HMI tags "2935RS001A01T05"
   "2935RS001A01T05.MSW" : 52809b66-421d-457f-8884-6f7a49d4e247 AT %DB5081.DBX18.0, 500 ms
   "2935RS001A01T05.DefaultText" : TextRef, internal   // Заголовок POPUP окна. При експорте из ECS через скрипт заполняется автоматически, если теги копируются в ручную то требуется в ручную задатать свойство Start Value
   "2935RS001A01T05.BlockInfo" : Array [0..2] of Int AT %DB5081.DBX38.0, 500 ms
   "2935RS001A01T05.StatusWork" : Int AT %DB5081.DBW242, 500 ms
   "2935RS001A01T05.FP_PARAM.DampingTime" : Int AT %DB5081.DBW50, 500 ms
   "2935RS001A01T05.FP_PARAM.Force_Value" : Real AT %DB5081.DBD52, 500 ms
   "2935RS001A01T05.FP_PARAM.Scale_Min" : Real AT %DB5081.DBD56, 500 ms
   "2935RS001A01T05.FP_PARAM.Scale_Max" : Real AT %DB5081.DBD60, 500 ms
   "2935RS001A01T05.FP_PARAM.Gradient" : Real AT %DB5081.DBD64, 500 ms
   "2935RS001A01T05.FP_PARAM.Grad_Pos" : Real AT %DB5081.DBD68, 500 ms
   "2935RS001A01T05.FP_PARAM.Grad_Neg" : Real AT %DB5081.DBD72, 500 ms
   "2935RS001A01T05.FP_PARAM.Grad_X" : Real AT %DB5081.DBD76, 500 ms
   "2935RS001A01T05.FP_PARAM.Gradient_Time_Pre" : Int AT %DB5081.DBW80, 500 ms
   "2935RS001A01T05.FP_PARAM.Gradient_Time_ACC" : Int AT %DB5081.DBW82, 500 ms
   "2935RS001A01T05.FP_PARAM.Alarm_Hyst" : Real AT %DB5081.DBD84, 500 ms
   "2935RS001A01T05.FP_PARAM.AlarmLimit_H3" : Real AT %DB5081.DBD88, 500 ms
   "2935RS001A01T05.FP_PARAM.AlarmLimit_H2" : Real AT %DB5081.DBD92, 500 ms
   "2935RS001A01T05.FP_PARAM.AlarmLimit_H1" : Real AT %DB5081.DBD96, 500 ms
   "2935RS001A01T05.FP_PARAM.AlarmLimit_L1" : Real AT %DB5081.DBD100, 500 ms
   "2935RS001A01T05.FP_PARAM.AlarmLimit_L2" : Real AT %DB5081.DBD104, 500 ms
   "2935RS001A01T05.FP_PARAM.AlarmLimit_L3" : Real AT %DB5081.DBD108, 500 ms
   "2935RS001A01T05.FP_PARAM.AlarmDelay_H3_Pre" : Int AT %DB5081.DBW112, 500 ms
   "2935RS001A01T05.FP_PARAM.AlarmDelay_H3_Acc" : Int AT %DB5081.DBW114, 500 ms
   "2935RS001A01T05.FP_PARAM.AlarmDelay_H2_Pre" : Int AT %DB5081.DBW116, 500 ms
   "2935RS001A01T05.FP_PARAM.AlarmDelay_H2_Acc" : Int AT %DB5081.DBW118, 500 ms
   "2935RS001A01T05.FP_PARAM.AlarmDelay_H1_Pre" : Int AT %DB5081.DBW120, 500 ms
   "2935RS001A01T05.FP_PARAM.AlarmDelay_H1_Acc" : Int AT %DB5081.DBW122, 500 ms
   "2935RS001A01T05.FP_PARAM.AlarmDelay_L1_Pre" : Int AT %DB5081.DBW124, 500 ms
   "2935RS001A01T05.FP_PARAM.AlarmDelay_L1_Acc" : Int AT %DB5081.DBW126, 500 ms
   "2935RS001A01T05.FP_PARAM.AlarmDelay_L2_Pre" : Int AT %DB5081.DBW128, 500 ms
   "2935RS001A01T05.FP_PARAM.AlarmDelay_L2_Acc" : Int AT %DB5081.DBW130, 500 ms
   "2935RS001A01T05.FP_PARAM.AlarmDelay_L3_Pre" : Int AT %DB5081.DBW132, 500 ms
   "2935RS001A01T05.FP_PARAM.AlarmDelay_L3_Acc" : Int AT %DB5081.DBW134, 500 ms
   "2935RS001A01T05.FP_PARAM.OpenLoopDelay_Pre" : Int AT %DB5081.DBW136, 500 ms
   "2935RS001A01T05.FP_PARAM.OpenLoopDelay_Acc" : Int AT %DB5081.DBW138, 500 ms
   "2935RS001A01T05.FP_PARAM.OverRangeDelay_Pre" : Int AT %DB5081.DBW140, 500 ms
   "2935RS001A01T05.FP_PARAM.OverRangeDelay_Acc" : Int AT %DB5081.DBW142, 500 ms
   "2935RS001A01T05.FP_PARAM.AuxLimit_H2_Value" : Real AT %DB5081.DBD144, 500 ms
   "2935RS001A01T05.FP_PARAM.AuxLimit_H1_Value" : Real AT %DB5081.DBD148, 500 ms
   "2935RS001A01T05.FP_PARAM.AuxLimit_L2_Value" : Real AT %DB5081.DBD152, 500 ms
   "2935RS001A01T05.FP_PARAM.AuxLimit_L1_Value" : Real AT %DB5081.DBD156, 500 ms
   "2935RS001A01T05.Unit" : TextRef, internal   // Еденицы измерения При експорте из ECS через скрипт заполняется автоматически, если теги копируются в ручную то требуется задатать свойство Text
   "2935RS001A01T05.Decimals" : TextRef, internal   // Формат отображения При експорте из ECS через скрипт, заполняется автоматически. Если теги копируются в ручную то требуется задатать свойство Text s999999.9
   "2935RS001A01T05.FP_EN.Square" : Bool AT %DB5081.DBX46.0, 500 ms
   "2935RS001A01T05.FP_EN.SquareRoot" : Bool AT %DB5081.DBX46.1, 500 ms
   "2935RS001A01T05.FP_EN.ParentSupress" : Bool AT %DB5081.DBX46.2, 500 ms
   "2935RS001A01T05.FP_EN.ParentSupressUnit" : Bool AT %DB5081.DBX46.3, 500 ms
   "2935RS001A01T05.FP_EN.Force" : Bool AT %DB5081.DBX46.4, 500 ms
   "2935RS001A01T05.FP_EN.Damping" : Bool AT %DB5081.DBX46.5, 500 ms
   "2935RS001A01T05.FP_EN.Gradient_Pos" : Bool AT %DB5081.DBX46.6, 500 ms
   "2935RS001A01T05.FP_EN.Gradient_Neg" : Bool AT %DB5081.DBX46.7, 500 ms
   "2935RS001A01T05.FP_EN.Hysteresis" : Bool AT %DB5081.DBX47.0, 500 ms
   "2935RS001A01T05.FP_EN.Alarm_H3" : Bool AT %DB5081.DBX47.1, 500 ms
   "2935RS001A01T05.FP_EN.Alarm_H2" : Bool AT %DB5081.DBX47.2, 500 ms
   "2935RS001A01T05.FP_EN.Alarm_H1" : Bool AT %DB5081.DBX47.3, 500 ms
   "2935RS001A01T05.FP_EN.Alarm_L1" : Bool AT %DB5081.DBX47.4, 500 ms
   "2935RS001A01T05.FP_EN.Alarm_L2" : Bool AT %DB5081.DBX47.5, 500 ms
   "2935RS001A01T05.FP_EN.Alarm_L3" : Bool AT %DB5081.DBX47.6, 500 ms
   "2935RS001A01T05.FP_EN.AlarmDelay_H3" : Bool AT %DB5081.DBX47.7, 500 ms
   "2935RS001A01T05.FP_EN.AlarmDelay_H2" : Bool AT %DB5081.DBX48.0, 500 ms
   "2935RS001A01T05.FP_EN.AlarmDelay_H1" : Bool AT %DB5081.DBX48.1, 500 ms
   "2935RS001A01T05.FP_EN.AlarmDelay_L1" : Bool AT %DB5081.DBX48.2, 500 ms
   "2935RS001A01T05.FP_EN.AlarmDelay_L2" : Bool AT %DB5081.DBX48.3, 500 ms
   "2935RS001A01T05.FP_EN.AlarmDelay_L3" : Bool AT %DB5081.DBX48.4, 500 ms
   "2935RS001A01T05.FP_EN.ROC_Warn" : Bool AT %DB5081.DBX48.5, 500 ms
   "2935RS001A01T05.FP_EN.U_Range_Warn" : Bool AT %DB5081.DBX48.6, 500 ms
   "2935RS001A01T05.FP_EN.O_Range_Warn" : Bool AT %DB5081.DBX48.7, 500 ms
   "2935RS001A01T05.trend_tag_name" : TextRef, internal   // Еденицы измерения При експорте из ECS через скрипт - заполняется автоматически, если теги копируются в ручную то требуется задатать свойство Text - имя тега для тренда
   "2935RS001A01T05.DQ.AL_H3" : Bool AT %DB5081.DBX16.0, 500 ms
   "2935RS001A01T05.DQ.AL_H2" : Bool AT %DB5081.DBX16.1, 500 ms
   "2935RS001A01T05.DQ.AL_H1" : Bool AT %DB5081.DBX16.2, 500 ms
   "2935RS001A01T05.DQ.AL_L1" : Bool AT %DB5081.DBX16.3, 500 ms
   "2935RS001A01T05.DQ.AL_L2" : Bool AT %DB5081.DBX16.4, 500 ms
   "2935RS001A01T05.DQ.AL_L3" : Bool AT %DB5081.DBX16.5, 500 ms
   "2935RS001A01T05.DQ.SIG_OK" : Bool AT %DB5081.DBX16.6, 500 ms
   "2935RS001A01T05.DQ.LIM_H2" : Bool AT %DB5081.DBX16.7, 500 ms
   "2935RS001A01T05.DQ.LIM_H1" : Bool AT %DB5081.DBX17.0, 500 ms
   "2935RS001A01T05.DQ.LIM_L1" : Bool AT %DB5081.DBX17.1, 500 ms
   "2935RS001A01T05.DQ.LIM_L2" : Bool AT %DB5081.DBX17.2, 500 ms
   "2935RS001A01T05.DQ.GR_P" : Bool AT %DB5081.DBX17.3, 500 ms
   "2935RS001A01T05.DQ.GR_N" : Bool AT %DB5081.DBX17.4, 500 ms
   "2935RS001A01T05.I.IN" : Real AT %DB5081.DBD2, 500 ms
   "2935RS001A01T05.I.SIG_TYPE" : Int AT %DB5081.DBW0, 500 ms
   "2935RS001A01T05.I.FI_BUS" : Byte AT %DB5081.DBB6, 500 ms
   "2935RS001A01T05.DI.U_RANGE" : Bool AT %DB5081.DBX7.0, 500 ms
   "2935RS001A01T05.DI.O_RANGE" : Bool AT %DB5081.DBX7.1, 500 ms
   "2935RS001A01T05.DI.SIG_FAULT" : Bool AT %DB5081.DBX7.2, 500 ms
   "2935RS001A01T05.DI.EnConfig" : Bool AT %DB5081.DBX7.3, 500 ms
   "2935RS001A01T05.DI.AEN" : Bool AT %DB5081.DBX7.4, 500 ms
   "2935RS001A01T05.DI.AL_SUPR" : Bool AT %DB5081.DBX7.5, 500 ms
   "2935RS001A01T05.Q.PV_NORM" : Real AT %DB5081.DBD8, 500 ms
   "2935RS001A01T05.Q.PV_SCAL" : Real AT %DB5081.DBD12, 500 ms
   "2935RS001A01T05.ParentInfo" : TextRef, internal   // Имя родителя для попап окна, вкладка инфо. При експорте из ECS через скрипт заполняется автоматически, если теги копируются в ручную то требуется в ручную задатать свойство Start Value

HMI tags "2940RS001A01F01"
   "2940RS001A01F01.MSW" : 52809b66-421d-457f-8884-6f7a49d4e247 AT %DB5082.DBX18.0, 500 ms
   "2940RS001A01F01.DefaultText" : TextRef, internal   // Заголовок POPUP окна. При експорте из ECS через скрипт заполняется автоматически, если теги копируются в ручную то требуется в ручную задатать свойство Start Value
   "2940RS001A01F01.BlockInfo" : Array [0..2] of Int AT %DB5082.DBX38.0, 500 ms
   "2940RS001A01F01.StatusWork" : Int AT %DB5082.DBW242, 500 ms
   "2940RS001A01F01.FP_PARAM.DampingTime" : Int AT %DB5082.DBW50, 500 ms
   "2940RS001A01F01.FP_PARAM.Force_Value" : Real AT %DB5082.DBD52, 500 ms
   "2940RS001A01F01.FP_PARAM.Scale_Min" : Real AT %DB5082.DBD56, 500 ms
   "2940RS001A01F01.FP_PARAM.Scale_Max" : Real AT %DB5082.DBD60, 500 ms
   "2940RS001A01F01.FP_PARAM.Gradient" : Real AT %DB5082.DBD64, 500 ms
   "2940RS001A01F01.FP_PARAM.Grad_Pos" : Real AT %DB5082.DBD68, 500 ms
   "2940RS001A01F01.FP_PARAM.Grad_Neg" : Real AT %DB5082.DBD72, 500 ms
   "2940RS001A01F01.FP_PARAM.Grad_X" : Real AT %DB5082.DBD76, 500 ms
   "2940RS001A01F01.FP_PARAM.Gradient_Time_Pre" : Int AT %DB5082.DBW80, 500 ms
   "2940RS001A01F01.FP_PARAM.Gradient_Time_ACC" : Int AT %DB5082.DBW82, 500 ms
   "2940RS001A01F01.FP_PARAM.Alarm_Hyst" : Real AT %DB5082.DBD84, 500 ms
   "2940RS001A01F01.FP_PARAM.AlarmLimit_H3" : Real AT %DB5082.DBD88, 500 ms
   "2940RS001A01F01.FP_PARAM.AlarmLimit_H2" : Real AT %DB5082.DBD92, 500 ms
   "2940RS001A01F01.FP_PARAM.AlarmLimit_H1" : Real AT %DB5082.DBD96, 500 ms
   "2940RS001A01F01.FP_PARAM.AlarmLimit_L1" : Real AT %DB5082.DBD100, 500 ms
   "2940RS001A01F01.FP_PARAM.AlarmLimit_L2" : Real AT %DB5082.DBD104, 500 ms
   "2940RS001A01F01.FP_PARAM.AlarmLimit_L3" : Real AT %DB5082.DBD108, 500 ms
   "2940RS001A01F01.FP_PARAM.AlarmDelay_H3_Pre" : Int AT %DB5082.DBW112, 500 ms
   "2940RS001A01F01.FP_PARAM.AlarmDelay_H3_Acc" : Int AT %DB5082.DBW114, 500 ms
   "2940RS001A01F01.FP_PARAM.AlarmDelay_H2_Pre" : Int AT %DB5082.DBW116, 500 ms
   "2940RS001A01F01.FP_PARAM.AlarmDelay_H2_Acc" : Int AT %DB5082.DBW118, 500 ms
   "2940RS001A01F01.FP_PARAM.AlarmDelay_H1_Pre" : Int AT %DB5082.DBW120, 500 ms
   "2940RS001A01F01.FP_PARAM.AlarmDelay_H1_Acc" : Int AT %DB5082.DBW122, 500 ms
   "2940RS001A01F01.FP_PARAM.AlarmDelay_L1_Pre" : Int AT %DB5082.DBW124, 500 ms
   "2940RS001A01F01.FP_PARAM.AlarmDelay_L1_Acc" : Int AT %DB5082.DBW126, 500 ms
   "2940RS001A01F01.FP_PARAM.AlarmDelay_L2_Pre" : Int AT %DB5082.DBW128, 500 ms
   "2940RS001A01F01.FP_PARAM.AlarmDelay_L2_Acc" : Int AT %DB5082.DBW130, 500 ms
   "2940RS001A01F01.FP_PARAM.AlarmDelay_L3_Pre" : Int AT %DB5082.DBW132, 500 ms
   "2940RS001A01F01.FP_PARAM.AlarmDelay_L3_Acc" : Int AT %DB5082.DBW134, 500 ms
   "2940RS001A01F01.FP_PARAM.OpenLoopDelay_Pre" : Int AT %DB5082.DBW136, 500 ms
   "2940RS001A01F01.FP_PARAM.OpenLoopDelay_Acc" : Int AT %DB5082.DBW138, 500 ms
   "2940RS001A01F01.FP_PARAM.OverRangeDelay_Pre" : Int AT %DB5082.DBW140, 500 ms
   "2940RS001A01F01.FP_PARAM.OverRangeDelay_Acc" : Int AT %DB5082.DBW142, 500 ms
   "2940RS001A01F01.FP_PARAM.AuxLimit_H2_Value" : Real AT %DB5082.DBD144, 500 ms
   "2940RS001A01F01.FP_PARAM.AuxLimit_H1_Value" : Real AT %DB5082.DBD148, 500 ms
   "2940RS001A01F01.FP_PARAM.AuxLimit_L2_Value" : Real AT %DB5082.DBD152, 500 ms
   "2940RS001A01F01.FP_PARAM.AuxLimit_L1_Value" : Real AT %DB5082.DBD156, 500 ms
   "2940RS001A01F01.Unit" : TextRef, internal   // Еденицы измерения При експорте из ECS через скрипт заполняется автоматически, если теги копируются в ручную то требуется задатать свойство Text
   "2940RS001A01F01.Decimals" : TextRef, internal   // Формат отображения При експорте из ECS через скрипт, заполняется автоматически. Если теги копируются в ручную то требуется задатать свойство Text s999999.9
   "2940RS001A01F01.FP_EN.Square" : Bool AT %DB5082.DBX46.0, 500 ms
   "2940RS001A01F01.FP_EN.SquareRoot" : Bool AT %DB5082.DBX46.1, 500 ms
   "2940RS001A01F01.FP_EN.ParentSupress" : Bool AT %DB5082.DBX46.2, 500 ms
   "2940RS001A01F01.FP_EN.ParentSupressUnit" : Bool AT %DB5082.DBX46.3, 500 ms
   "2940RS001A01F01.FP_EN.Force" : Bool AT %DB5082.DBX46.4, 500 ms
   "2940RS001A01F01.FP_EN.Damping" : Bool AT %DB5082.DBX46.5, 500 ms
   "2940RS001A01F01.FP_EN.Gradient_Pos" : Bool AT %DB5082.DBX46.6, 500 ms
   "2940RS001A01F01.FP_EN.Gradient_Neg" : Bool AT %DB5082.DBX46.7, 500 ms
   "2940RS001A01F01.FP_EN.Hysteresis" : Bool AT %DB5082.DBX47.0, 500 ms
   "2940RS001A01F01.FP_EN.Alarm_H3" : Bool AT %DB5082.DBX47.1, 500 ms
   "2940RS001A01F01.FP_EN.Alarm_H2" : Bool AT %DB5082.DBX47.2, 500 ms
   "2940RS001A01F01.FP_EN.Alarm_H1" : Bool AT %DB5082.DBX47.3, 500 ms
   "2940RS001A01F01.FP_EN.Alarm_L1" : Bool AT %DB5082.DBX47.4, 500 ms
   "2940RS001A01F01.FP_EN.Alarm_L2" : Bool AT %DB5082.DBX47.5, 500 ms
   "2940RS001A01F01.FP_EN.Alarm_L3" : Bool AT %DB5082.DBX47.6, 500 ms
   "2940RS001A01F01.FP_EN.AlarmDelay_H3" : Bool AT %DB5082.DBX47.7, 500 ms
   "2940RS001A01F01.FP_EN.AlarmDelay_H2" : Bool AT %DB5082.DBX48.0, 500 ms
   "2940RS001A01F01.FP_EN.AlarmDelay_H1" : Bool AT %DB5082.DBX48.1, 500 ms
   "2940RS001A01F01.FP_EN.AlarmDelay_L1" : Bool AT %DB5082.DBX48.2, 500 ms
   "2940RS001A01F01.FP_EN.AlarmDelay_L2" : Bool AT %DB5082.DBX48.3, 500 ms
   "2940RS001A01F01.FP_EN.AlarmDelay_L3" : Bool AT %DB5082.DBX48.4, 500 ms
   "2940RS001A01F01.FP_EN.ROC_Warn" : Bool AT %DB5082.DBX48.5, 500 ms
   "2940RS001A01F01.FP_EN.U_Range_Warn" : Bool AT %DB5082.DBX48.6, 500 ms
   "2940RS001A01F01.FP_EN.O_Range_Warn" : Bool AT %DB5082.DBX48.7, 500 ms
   "2940RS001A01F01.trend_tag_name" : TextRef, internal   // Еденицы измерения При експорте из ECS через скрипт - заполняется автоматически, если теги копируются в ручную то требуется задатать свойство Text - имя тега для тренда
   "2940RS001A01F01.DQ.AL_H3" : Bool AT %DB5082.DBX16.0, 500 ms
   "2940RS001A01F01.DQ.AL_H2" : Bool AT %DB5082.DBX16.1, 500 ms
   "2940RS001A01F01.DQ.AL_H1" : Bool AT %DB5082.DBX16.2, 500 ms
   "2940RS001A01F01.DQ.AL_L1" : Bool AT %DB5082.DBX16.3, 500 ms
   "2940RS001A01F01.DQ.AL_L2" : Bool AT %DB5082.DBX16.4, 500 ms
   "2940RS001A01F01.DQ.AL_L3" : Bool AT %DB5082.DBX16.5, 500 ms
   "2940RS001A01F01.DQ.SIG_OK" : Bool AT %DB5082.DBX16.6, 500 ms
   "2940RS001A01F01.DQ.LIM_H2" : Bool AT %DB5082.DBX16.7, 500 ms
   "2940RS001A01F01.DQ.LIM_H1" : Bool AT %DB5082.DBX17.0, 500 ms
   "2940RS001A01F01.DQ.LIM_L1" : Bool AT %DB5082.DBX17.1, 500 ms
   "2940RS001A01F01.DQ.LIM_L2" : Bool AT %DB5082.DBX17.2, 500 ms
   "2940RS001A01F01.DQ.GR_P" : Bool AT %DB5082.DBX17.3, 500 ms
   "2940RS001A01F01.DQ.GR_N" : Bool AT %DB5082.DBX17.4, 500 ms
   "2940RS001A01F01.I.IN" : Real AT %DB5082.DBD2, 500 ms
   "2940RS001A01F01.I.SIG_TYPE" : Int AT %DB5082.DBW0, 500 ms
   "2940RS001A01F01.I.FI_BUS" : Byte AT %DB5082.DBB6, 500 ms
   "2940RS001A01F01.DI.U_RANGE" : Bool AT %DB5082.DBX7.0, 500 ms
   "2940RS001A01F01.DI.O_RANGE" : Bool AT %DB5082.DBX7.1, 500 ms
   "2940RS001A01F01.DI.SIG_FAULT" : Bool AT %DB5082.DBX7.2, 500 ms
   "2940RS001A01F01.DI.EnConfig" : Bool AT %DB5082.DBX7.3, 500 ms
   "2940RS001A01F01.DI.AEN" : Bool AT %DB5082.DBX7.4, 500 ms
   "2940RS001A01F01.DI.AL_SUPR" : Bool AT %DB5082.DBX7.5, 500 ms
   "2940RS001A01F01.Q.PV_NORM" : Real AT %DB5082.DBD8, 500 ms
   "2940RS001A01F01.Q.PV_SCAL" : Real AT %DB5082.DBD12, 500 ms
   "2940RS001A01F01.ParentInfo" : TextRef, internal   // Имя родителя для попап окна, вкладка инфо. При експорте из ECS через скрипт заполняется автоматически, если теги копируются в ручную то требуется в ручную задатать свойство Start Value

HMI tags "2940RS001A01L01"
   "2940RS001A01L01.MSW" : 52809b66-421d-457f-8884-6f7a49d4e247 AT %DB5083.DBX18.0, 500 ms
   "2940RS001A01L01.DefaultText" : TextRef, internal   // Заголовок POPUP окна. При експорте из ECS через скрипт заполняется автоматически, если теги копируются в ручную то требуется в ручную задатать свойство Start Value
   "2940RS001A01L01.BlockInfo" : Array [0..2] of Int AT %DB5083.DBX38.0, 500 ms
   "2940RS001A01L01.StatusWork" : Int AT %DB5083.DBW242, 500 ms
   "2940RS001A01L01.FP_PARAM.DampingTime" : Int AT %DB5083.DBW50, 500 ms
   "2940RS001A01L01.FP_PARAM.Force_Value" : Real AT %DB5083.DBD52, 500 ms
   "2940RS001A01L01.FP_PARAM.Scale_Min" : Real AT %DB5083.DBD56, 500 ms
   "2940RS001A01L01.FP_PARAM.Scale_Max" : Real AT %DB5083.DBD60, 500 ms
   "2940RS001A01L01.FP_PARAM.Gradient" : Real AT %DB5083.DBD64, 500 ms
   "2940RS001A01L01.FP_PARAM.Grad_Pos" : Real AT %DB5083.DBD68, 500 ms
   "2940RS001A01L01.FP_PARAM.Grad_Neg" : Real AT %DB5083.DBD72, 500 ms
   "2940RS001A01L01.FP_PARAM.Grad_X" : Real AT %DB5083.DBD76, 500 ms
   "2940RS001A01L01.FP_PARAM.Gradient_Time_Pre" : Int AT %DB5083.DBW80, 500 ms
   "2940RS001A01L01.FP_PARAM.Gradient_Time_ACC" : Int AT %DB5083.DBW82, 500 ms
   "2940RS001A01L01.FP_PARAM.Alarm_Hyst" : Real AT %DB5083.DBD84, 500 ms
   "2940RS001A01L01.FP_PARAM.AlarmLimit_H3" : Real AT %DB5083.DBD88, 500 ms
   "2940RS001A01L01.FP_PARAM.AlarmLimit_H2" : Real AT %DB5083.DBD92, 500 ms
   "2940RS001A01L01.FP_PARAM.AlarmLimit_H1" : Real AT %DB5083.DBD96, 500 ms
   "2940RS001A01L01.FP_PARAM.AlarmLimit_L1" : Real AT %DB5083.DBD100, 500 ms
   "2940RS001A01L01.FP_PARAM.AlarmLimit_L2" : Real AT %DB5083.DBD104, 500 ms
   "2940RS001A01L01.FP_PARAM.AlarmLimit_L3" : Real AT %DB5083.DBD108, 500 ms
   "2940RS001A01L01.FP_PARAM.AlarmDelay_H3_Pre" : Int AT %DB5083.DBW112, 500 ms
   "2940RS001A01L01.FP_PARAM.AlarmDelay_H3_Acc" : Int AT %DB5083.DBW114, 500 ms
   "2940RS001A01L01.FP_PARAM.AlarmDelay_H2_Pre" : Int AT %DB5083.DBW116, 500 ms
   "2940RS001A01L01.FP_PARAM.AlarmDelay_H2_Acc" : Int AT %DB5083.DBW118, 500 ms
   "2940RS001A01L01.FP_PARAM.AlarmDelay_H1_Pre" : Int AT %DB5083.DBW120, 500 ms
   "2940RS001A01L01.FP_PARAM.AlarmDelay_H1_Acc" : Int AT %DB5083.DBW122, 500 ms
   "2940RS001A01L01.FP_PARAM.AlarmDelay_L1_Pre" : Int AT %DB5083.DBW124, 500 ms
   "2940RS001A01L01.FP_PARAM.AlarmDelay_L1_Acc" : Int AT %DB5083.DBW126, 500 ms
   "2940RS001A01L01.FP_PARAM.AlarmDelay_L2_Pre" : Int AT %DB5083.DBW128, 500 ms
   "2940RS001A01L01.FP_PARAM.AlarmDelay_L2_Acc" : Int AT %DB5083.DBW130, 500 ms
   "2940RS001A01L01.FP_PARAM.AlarmDelay_L3_Pre" : Int AT %DB5083.DBW132, 500 ms
   "2940RS001A01L01.FP_PARAM.AlarmDelay_L3_Acc" : Int AT %DB5083.DBW134, 500 ms
   "2940RS001A01L01.FP_PARAM.OpenLoopDelay_Pre" : Int AT %DB5083.DBW136, 500 ms
   "2940RS001A01L01.FP_PARAM.OpenLoopDelay_Acc" : Int AT %DB5083.DBW138, 500 ms
   "2940RS001A01L01.FP_PARAM.OverRangeDelay_Pre" : Int AT %DB5083.DBW140, 500 ms
   "2940RS001A01L01.FP_PARAM.OverRangeDelay_Acc" : Int AT %DB5083.DBW142, 500 ms
   "2940RS001A01L01.FP_PARAM.AuxLimit_H2_Value" : Real AT %DB5083.DBD144, 500 ms
   "2940RS001A01L01.FP_PARAM.AuxLimit_H1_Value" : Real AT %DB5083.DBD148, 500 ms
   "2940RS001A01L01.FP_PARAM.AuxLimit_L2_Value" : Real AT %DB5083.DBD152, 500 ms
   "2940RS001A01L01.FP_PARAM.AuxLimit_L1_Value" : Real AT %DB5083.DBD156, 500 ms
   "2940RS001A01L01.Unit" : TextRef, internal   // Еденицы измерения При експорте из ECS через скрипт заполняется автоматически, если теги копируются в ручную то требуется задатать свойство Text
   "2940RS001A01L01.Decimals" : TextRef, internal   // Формат отображения При експорте из ECS через скрипт, заполняется автоматически. Если теги копируются в ручную то требуется задатать свойство Text s999999.9
   "2940RS001A01L01.FP_EN.Square" : Bool AT %DB5083.DBX46.0, 500 ms
   "2940RS001A01L01.FP_EN.SquareRoot" : Bool AT %DB5083.DBX46.1, 500 ms
   "2940RS001A01L01.FP_EN.ParentSupress" : Bool AT %DB5083.DBX46.2, 500 ms
   "2940RS001A01L01.FP_EN.ParentSupressUnit" : Bool AT %DB5083.DBX46.3, 500 ms
   "2940RS001A01L01.FP_EN.Force" : Bool AT %DB5083.DBX46.4, 500 ms
   "2940RS001A01L01.FP_EN.Damping" : Bool AT %DB5083.DBX46.5, 500 ms
   "2940RS001A01L01.FP_EN.Gradient_Pos" : Bool AT %DB5083.DBX46.6, 500 ms
   "2940RS001A01L01.FP_EN.Gradient_Neg" : Bool AT %DB5083.DBX46.7, 500 ms
   "2940RS001A01L01.FP_EN.Hysteresis" : Bool AT %DB5083.DBX47.0, 500 ms
   "2940RS001A01L01.FP_EN.Alarm_H3" : Bool AT %DB5083.DBX47.1, 500 ms
   "2940RS001A01L01.FP_EN.Alarm_H2" : Bool AT %DB5083.DBX47.2, 500 ms
   "2940RS001A01L01.FP_EN.Alarm_H1" : Bool AT %DB5083.DBX47.3, 500 ms
   "2940RS001A01L01.FP_EN.Alarm_L1" : Bool AT %DB5083.DBX47.4, 500 ms
   "2940RS001A01L01.FP_EN.Alarm_L2" : Bool AT %DB5083.DBX47.5, 500 ms
   "2940RS001A01L01.FP_EN.Alarm_L3" : Bool AT %DB5083.DBX47.6, 500 ms
   "2940RS001A01L01.FP_EN.AlarmDelay_H3" : Bool AT %DB5083.DBX47.7, 500 ms
   "2940RS001A01L01.FP_EN.AlarmDelay_H2" : Bool AT %DB5083.DBX48.0, 500 ms
   "2940RS001A01L01.FP_EN.AlarmDelay_H1" : Bool AT %DB5083.DBX48.1, 500 ms
   "2940RS001A01L01.FP_EN.AlarmDelay_L1" : Bool AT %DB5083.DBX48.2, 500 ms
   "2940RS001A01L01.FP_EN.AlarmDelay_L2" : Bool AT %DB5083.DBX48.3, 500 ms
   "2940RS001A01L01.FP_EN.AlarmDelay_L3" : Bool AT %DB5083.DBX48.4, 500 ms
   "2940RS001A01L01.FP_EN.ROC_Warn" : Bool AT %DB5083.DBX48.5, 500 ms
   "2940RS001A01L01.FP_EN.U_Range_Warn" : Bool AT %DB5083.DBX48.6, 500 ms
   "2940RS001A01L01.FP_EN.O_Range_Warn" : Bool AT %DB5083.DBX48.7, 500 ms
   "2940RS001A01L01.trend_tag_name" : TextRef, internal   // Еденицы измерения При експорте из ECS через скрипт - заполняется автоматически, если теги копируются в ручную то требуется задатать свойство Text - имя тега для тренда
   "2940RS001A01L01.DQ.AL_H3" : Bool AT %DB5083.DBX16.0, 500 ms
   "2940RS001A01L01.DQ.AL_H2" : Bool AT %DB5083.DBX16.1, 500 ms
   "2940RS001A01L01.DQ.AL_H1" : Bool AT %DB5083.DBX16.2, 500 ms
   "2940RS001A01L01.DQ.AL_L1" : Bool AT %DB5083.DBX16.3, 500 ms
   "2940RS001A01L01.DQ.AL_L2" : Bool AT %DB5083.DBX16.4, 500 ms
   "2940RS001A01L01.DQ.AL_L3" : Bool AT %DB5083.DBX16.5, 500 ms
   "2940RS001A01L01.DQ.SIG_OK" : Bool AT %DB5083.DBX16.6, 500 ms
   "2940RS001A01L01.DQ.LIM_H2" : Bool AT %DB5083.DBX16.7, 500 ms
   "2940RS001A01L01.DQ.LIM_H1" : Bool AT %DB5083.DBX17.0, 500 ms
   "2940RS001A01L01.DQ.LIM_L1" : Bool AT %DB5083.DBX17.1, 500 ms
   "2940RS001A01L01.DQ.LIM_L2" : Bool AT %DB5083.DBX17.2, 500 ms
   "2940RS001A01L01.DQ.GR_P" : Bool AT %DB5083.DBX17.3, 500 ms
   "2940RS001A01L01.DQ.GR_N" : Bool AT %DB5083.DBX17.4, 500 ms
   "2940RS001A01L01.I.IN" : Real AT %DB5083.DBD2, 500 ms
   "2940RS001A01L01.I.SIG_TYPE" : Int AT %DB5083.DBW0, 500 ms
   "2940RS001A01L01.I.FI_BUS" : Byte AT %DB5083.DBB6, 500 ms
   "2940RS001A01L01.DI.U_RANGE" : Bool AT %DB5083.DBX7.0, 500 ms
   "2940RS001A01L01.DI.O_RANGE" : Bool AT %DB5083.DBX7.1, 500 ms
   "2940RS001A01L01.DI.SIG_FAULT" : Bool AT %DB5083.DBX7.2, 500 ms
   "2940RS001A01L01.DI.EnConfig" : Bool AT %DB5083.DBX7.3, 500 ms
   "2940RS001A01L01.DI.AEN" : Bool AT %DB5083.DBX7.4, 500 ms
   "2940RS001A01L01.DI.AL_SUPR" : Bool AT %DB5083.DBX7.5, 500 ms
   "2940RS001A01L01.Q.PV_NORM" : Real AT %DB5083.DBD8, 500 ms
   "2940RS001A01L01.Q.PV_SCAL" : Real AT %DB5083.DBD12, 500 ms
   "2940RS001A01L01.ParentInfo" : TextRef, internal   // Имя родителя для попап окна, вкладка инфо. При експорте из ECS через скрипт заполняется автоматически, если теги копируются в ручную то требуется в ручную задатать свойство Start Value

HMI tags "2940RS001A01T01"
   "2940RS001A01T01.MSW" : 52809b66-421d-457f-8884-6f7a49d4e247 AT %DB5084.DBX18.0, 500 ms
   "2940RS001A01T01.DefaultText" : TextRef, internal   // Заголовок POPUP окна. При експорте из ECS через скрипт заполняется автоматически, если теги копируются в ручную то требуется в ручную задатать свойство Start Value
   "2940RS001A01T01.BlockInfo" : Array [0..2] of Int AT %DB5084.DBX38.0, 500 ms
   "2940RS001A01T01.StatusWork" : Int AT %DB5084.DBW242, 500 ms
   "2940RS001A01T01.FP_PARAM.DampingTime" : Int AT %DB5084.DBW50, 500 ms
   "2940RS001A01T01.FP_PARAM.Force_Value" : Real AT %DB5084.DBD52, 500 ms
   "2940RS001A01T01.FP_PARAM.Scale_Min" : Real AT %DB5084.DBD56, 500 ms
   "2940RS001A01T01.FP_PARAM.Scale_Max" : Real AT %DB5084.DBD60, 500 ms
   "2940RS001A01T01.FP_PARAM.Gradient" : Real AT %DB5084.DBD64, 500 ms
   "2940RS001A01T01.FP_PARAM.Grad_Pos" : Real AT %DB5084.DBD68, 500 ms
   "2940RS001A01T01.FP_PARAM.Grad_Neg" : Real AT %DB5084.DBD72, 500 ms
   "2940RS001A01T01.FP_PARAM.Grad_X" : Real AT %DB5084.DBD76, 500 ms
   "2940RS001A01T01.FP_PARAM.Gradient_Time_Pre" : Int AT %DB5084.DBW80, 500 ms
   "2940RS001A01T01.FP_PARAM.Gradient_Time_ACC" : Int AT %DB5084.DBW82, 500 ms
   "2940RS001A01T01.FP_PARAM.Alarm_Hyst" : Real AT %DB5084.DBD84, 500 ms
   "2940RS001A01T01.FP_PARAM.AlarmLimit_H3" : Real AT %DB5084.DBD88, 500 ms
   "2940RS001A01T01.FP_PARAM.AlarmLimit_H2" : Real AT %DB5084.DBD92, 500 ms
   "2940RS001A01T01.FP_PARAM.AlarmLimit_H1" : Real AT %DB5084.DBD96, 500 ms
   "2940RS001A01T01.FP_PARAM.AlarmLimit_L1" : Real AT %DB5084.DBD100, 500 ms
   "2940RS001A01T01.FP_PARAM.AlarmLimit_L2" : Real AT %DB5084.DBD104, 500 ms
   "2940RS001A01T01.FP_PARAM.AlarmLimit_L3" : Real AT %DB5084.DBD108, 500 ms
   "2940RS001A01T01.FP_PARAM.AlarmDelay_H3_Pre" : Int AT %DB5084.DBW112, 500 ms
   "2940RS001A01T01.FP_PARAM.AlarmDelay_H3_Acc" : Int AT %DB5084.DBW114, 500 ms
   "2940RS001A01T01.FP_PARAM.AlarmDelay_H2_Pre" : Int AT %DB5084.DBW116, 500 ms
   "2940RS001A01T01.FP_PARAM.AlarmDelay_H2_Acc" : Int AT %DB5084.DBW118, 500 ms
   "2940RS001A01T01.FP_PARAM.AlarmDelay_H1_Pre" : Int AT %DB5084.DBW120, 500 ms
   "2940RS001A01T01.FP_PARAM.AlarmDelay_H1_Acc" : Int AT %DB5084.DBW122, 500 ms
   "2940RS001A01T01.FP_PARAM.AlarmDelay_L1_Pre" : Int AT %DB5084.DBW124, 500 ms
   "2940RS001A01T01.FP_PARAM.AlarmDelay_L1_Acc" : Int AT %DB5084.DBW126, 500 ms
   "2940RS001A01T01.FP_PARAM.AlarmDelay_L2_Pre" : Int AT %DB5084.DBW128, 500 ms
   "2940RS001A01T01.FP_PARAM.AlarmDelay_L2_Acc" : Int AT %DB5084.DBW130, 500 ms
   "2940RS001A01T01.FP_PARAM.AlarmDelay_L3_Pre" : Int AT %DB5084.DBW132, 500 ms
   "2940RS001A01T01.FP_PARAM.AlarmDelay_L3_Acc" : Int AT %DB5084.DBW134, 500 ms
   "2940RS001A01T01.FP_PARAM.OpenLoopDelay_Pre" : Int AT %DB5084.DBW136, 500 ms
   "2940RS001A01T01.FP_PARAM.OpenLoopDelay_Acc" : Int AT %DB5084.DBW138, 500 ms
   "2940RS001A01T01.FP_PARAM.OverRangeDelay_Pre" : Int AT %DB5084.DBW140, 500 ms
   "2940RS001A01T01.FP_PARAM.OverRangeDelay_Acc" : Int AT %DB5084.DBW142, 500 ms
   "2940RS001A01T01.FP_PARAM.AuxLimit_H2_Value" : Real AT %DB5084.DBD144, 500 ms
   "2940RS001A01T01.FP_PARAM.AuxLimit_H1_Value" : Real AT %DB5084.DBD148, 500 ms
   "2940RS001A01T01.FP_PARAM.AuxLimit_L2_Value" : Real AT %DB5084.DBD152, 500 ms
   "2940RS001A01T01.FP_PARAM.AuxLimit_L1_Value" : Real AT %DB5084.DBD156, 500 ms
   "2940RS001A01T01.Unit" : TextRef, internal   // Еденицы измерения При експорте из ECS через скрипт заполняется автоматически, если теги копируются в ручную то требуется задатать свойство Text
   "2940RS001A01T01.Decimals" : TextRef, internal   // Формат отображения При експорте из ECS через скрипт, заполняется автоматически. Если теги копируются в ручную то требуется задатать свойство Text s999999.9
   "2940RS001A01T01.FP_EN.Square" : Bool AT %DB5084.DBX46.0, 500 ms
   "2940RS001A01T01.FP_EN.SquareRoot" : Bool AT %DB5084.DBX46.1, 500 ms
   "2940RS001A01T01.FP_EN.ParentSupress" : Bool AT %DB5084.DBX46.2, 500 ms
   "2940RS001A01T01.FP_EN.ParentSupressUnit" : Bool AT %DB5084.DBX46.3, 500 ms
   "2940RS001A01T01.FP_EN.Force" : Bool AT %DB5084.DBX46.4, 500 ms
   "2940RS001A01T01.FP_EN.Damping" : Bool AT %DB5084.DBX46.5, 500 ms
   "2940RS001A01T01.FP_EN.Gradient_Pos" : Bool AT %DB5084.DBX46.6, 500 ms
   "2940RS001A01T01.FP_EN.Gradient_Neg" : Bool AT %DB5084.DBX46.7, 500 ms
   "2940RS001A01T01.FP_EN.Hysteresis" : Bool AT %DB5084.DBX47.0, 500 ms
   "2940RS001A01T01.FP_EN.Alarm_H3" : Bool AT %DB5084.DBX47.1, 500 ms
   "2940RS001A01T01.FP_EN.Alarm_H2" : Bool AT %DB5084.DBX47.2, 500 ms
   "2940RS001A01T01.FP_EN.Alarm_H1" : Bool AT %DB5084.DBX47.3, 500 ms
   "2940RS001A01T01.FP_EN.Alarm_L1" : Bool AT %DB5084.DBX47.4, 500 ms
   "2940RS001A01T01.FP_EN.Alarm_L2" : Bool AT %DB5084.DBX47.5, 500 ms
   "2940RS001A01T01.FP_EN.Alarm_L3" : Bool AT %DB5084.DBX47.6, 500 ms
   "2940RS001A01T01.FP_EN.AlarmDelay_H3" : Bool AT %DB5084.DBX47.7, 500 ms
   "2940RS001A01T01.FP_EN.AlarmDelay_H2" : Bool AT %DB5084.DBX48.0, 500 ms
   "2940RS001A01T01.FP_EN.AlarmDelay_H1" : Bool AT %DB5084.DBX48.1, 500 ms
   "2940RS001A01T01.FP_EN.AlarmDelay_L1" : Bool AT %DB5084.DBX48.2, 500 ms
   "2940RS001A01T01.FP_EN.AlarmDelay_L2" : Bool AT %DB5084.DBX48.3, 500 ms
   "2940RS001A01T01.FP_EN.AlarmDelay_L3" : Bool AT %DB5084.DBX48.4, 500 ms
   "2940RS001A01T01.FP_EN.ROC_Warn" : Bool AT %DB5084.DBX48.5, 500 ms
   "2940RS001A01T01.FP_EN.U_Range_Warn" : Bool AT %DB5084.DBX48.6, 500 ms
   "2940RS001A01T01.FP_EN.O_Range_Warn" : Bool AT %DB5084.DBX48.7, 500 ms
   "2940RS001A01T01.trend_tag_name" : TextRef, internal   // Еденицы измерения При експорте из ECS через скрипт - заполняется автоматически, если теги копируются в ручную то требуется задатать свойство Text - имя тега для тренда
   "2940RS001A01T01.DQ.AL_H3" : Bool AT %DB5084.DBX16.0, 500 ms
   "2940RS001A01T01.DQ.AL_H2" : Bool AT %DB5084.DBX16.1, 500 ms
   "2940RS001A01T01.DQ.AL_H1" : Bool AT %DB5084.DBX16.2, 500 ms
   "2940RS001A01T01.DQ.AL_L1" : Bool AT %DB5084.DBX16.3, 500 ms
   "2940RS001A01T01.DQ.AL_L2" : Bool AT %DB5084.DBX16.4, 500 ms
   "2940RS001A01T01.DQ.AL_L3" : Bool AT %DB5084.DBX16.5, 500 ms
   "2940RS001A01T01.DQ.SIG_OK" : Bool AT %DB5084.DBX16.6, 500 ms
   "2940RS001A01T01.DQ.LIM_H2" : Bool AT %DB5084.DBX16.7, 500 ms
   "2940RS001A01T01.DQ.LIM_H1" : Bool AT %DB5084.DBX17.0, 500 ms
   "2940RS001A01T01.DQ.LIM_L1" : Bool AT %DB5084.DBX17.1, 500 ms
   "2940RS001A01T01.DQ.LIM_L2" : Bool AT %DB5084.DBX17.2, 500 ms
   "2940RS001A01T01.DQ.GR_P" : Bool AT %DB5084.DBX17.3, 500 ms
   "2940RS001A01T01.DQ.GR_N" : Bool AT %DB5084.DBX17.4, 500 ms
   "2940RS001A01T01.I.IN" : Real AT %DB5084.DBD2, 500 ms
   "2940RS001A01T01.I.SIG_TYPE" : Int AT %DB5084.DBW0, 500 ms
   "2940RS001A01T01.I.FI_BUS" : Byte AT %DB5084.DBB6, 500 ms
   "2940RS001A01T01.DI.U_RANGE" : Bool AT %DB5084.DBX7.0, 500 ms
   "2940RS001A01T01.DI.O_RANGE" : Bool AT %DB5084.DBX7.1, 500 ms
   "2940RS001A01T01.DI.SIG_FAULT" : Bool AT %DB5084.DBX7.2, 500 ms
   "2940RS001A01T01.DI.EnConfig" : Bool AT %DB5084.DBX7.3, 500 ms
   "2940RS001A01T01.DI.AEN" : Bool AT %DB5084.DBX7.4, 500 ms
   "2940RS001A01T01.DI.AL_SUPR" : Bool AT %DB5084.DBX7.5, 500 ms
   "2940RS001A01T01.Q.PV_NORM" : Real AT %DB5084.DBD8, 500 ms
   "2940RS001A01T01.Q.PV_SCAL" : Real AT %DB5084.DBD12, 500 ms
   "2940RS001A01T01.ParentInfo" : TextRef, internal   // Имя родителя для попап окна, вкладка инфо. При експорте из ECS через скрипт заполняется автоматически, если теги копируются в ручную то требуется в ручную задатать свойство Start Value

HMI tags "2940RS001N01T01"
   "2940RS001N01T01.MSW" : 52809b66-421d-457f-8884-6f7a49d4e247 AT %DB5304.DBX18.0, 500 ms
   "2940RS001N01T01.DefaultText" : TextRef, internal   // Заголовок POPUP окна. При експорте из ECS через скрипт заполняется автоматически, если теги копируются в ручную то требуется в ручную задатать свойство Start Value
   "2940RS001N01T01.BlockInfo" : Array [0..2] of Int AT %DB5304.DBX38.0, 500 ms
   "2940RS001N01T01.StatusWork" : Int AT %DB5304.DBW242, 500 ms
   "2940RS001N01T01.FP_PARAM.DampingTime" : Int AT %DB5304.DBW50, 500 ms
   "2940RS001N01T01.FP_PARAM.Force_Value" : Real AT %DB5304.DBD52, 500 ms
   "2940RS001N01T01.FP_PARAM.Scale_Min" : Real AT %DB5304.DBD56, 500 ms
   "2940RS001N01T01.FP_PARAM.Scale_Max" : Real AT %DB5304.DBD60, 500 ms
   "2940RS001N01T01.FP_PARAM.Gradient" : Real AT %DB5304.DBD64, 500 ms
   "2940RS001N01T01.FP_PARAM.Grad_Pos" : Real AT %DB5304.DBD68, 500 ms
   "2940RS001N01T01.FP_PARAM.Grad_Neg" : Real AT %DB5304.DBD72, 500 ms
   "2940RS001N01T01.FP_PARAM.Grad_X" : Real AT %DB5304.DBD76, 500 ms
   "2940RS001N01T01.FP_PARAM.Gradient_Time_Pre" : Int AT %DB5304.DBW80, 500 ms
   "2940RS001N01T01.FP_PARAM.Gradient_Time_ACC" : Int AT %DB5304.DBW82, 500 ms
   "2940RS001N01T01.FP_PARAM.Alarm_Hyst" : Real AT %DB5304.DBD84, 500 ms
   "2940RS001N01T01.FP_PARAM.AlarmLimit_H3" : Real AT %DB5304.DBD88, 500 ms
   "2940RS001N01T01.FP_PARAM.AlarmLimit_H2" : Real AT %DB5304.DBD92, 500 ms
   "2940RS001N01T01.FP_PARAM.AlarmLimit_H1" : Real AT %DB5304.DBD96, 500 ms
   "2940RS001N01T01.FP_PARAM.AlarmLimit_L1" : Real AT %DB5304.DBD100, 500 ms
   "2940RS001N01T01.FP_PARAM.AlarmLimit_L2" : Real AT %DB5304.DBD104, 500 ms
   "2940RS001N01T01.FP_PARAM.AlarmLimit_L3" : Real AT %DB5304.DBD108, 500 ms
   "2940RS001N01T01.FP_PARAM.AlarmDelay_H3_Pre" : Int AT %DB5304.DBW112, 500 ms
   "2940RS001N01T01.FP_PARAM.AlarmDelay_H3_Acc" : Int AT %DB5304.DBW114, 500 ms
   "2940RS001N01T01.FP_PARAM.AlarmDelay_H2_Pre" : Int AT %DB5304.DBW116, 500 ms
   "2940RS001N01T01.FP_PARAM.AlarmDelay_H2_Acc" : Int AT %DB5304.DBW118, 500 ms
   "2940RS001N01T01.FP_PARAM.AlarmDelay_H1_Pre" : Int AT %DB5304.DBW120, 500 ms
   "2940RS001N01T01.FP_PARAM.AlarmDelay_H1_Acc" : Int AT %DB5304.DBW122, 500 ms
   "2940RS001N01T01.FP_PARAM.AlarmDelay_L1_Pre" : Int AT %DB5304.DBW124, 500 ms
   "2940RS001N01T01.FP_PARAM.AlarmDelay_L1_Acc" : Int AT %DB5304.DBW126, 500 ms
   "2940RS001N01T01.FP_PARAM.AlarmDelay_L2_Pre" : Int AT %DB5304.DBW128, 500 ms
   "2940RS001N01T01.FP_PARAM.AlarmDelay_L2_Acc" : Int AT %DB5304.DBW130, 500 ms
   "2940RS001N01T01.FP_PARAM.AlarmDelay_L3_Pre" : Int AT %DB5304.DBW132, 500 ms
   "2940RS001N01T01.FP_PARAM.AlarmDelay_L3_Acc" : Int AT %DB5304.DBW134, 500 ms
   "2940RS001N01T01.FP_PARAM.OpenLoopDelay_Pre" : Int AT %DB5304.DBW136, 500 ms
   "2940RS001N01T01.FP_PARAM.OpenLoopDelay_Acc" : Int AT %DB5304.DBW138, 500 ms
   "2940RS001N01T01.FP_PARAM.OverRangeDelay_Pre" : Int AT %DB5304.DBW140, 500 ms
   "2940RS001N01T01.FP_PARAM.OverRangeDelay_Acc" : Int AT %DB5304.DBW142, 500 ms
   "2940RS001N01T01.FP_PARAM.AuxLimit_H2_Value" : Real AT %DB5304.DBD144, 500 ms
   "2940RS001N01T01.FP_PARAM.AuxLimit_H1_Value" : Real AT %DB5304.DBD148, 500 ms
   "2940RS001N01T01.FP_PARAM.AuxLimit_L2_Value" : Real AT %DB5304.DBD152, 500 ms
   "2940RS001N01T01.FP_PARAM.AuxLimit_L1_Value" : Real AT %DB5304.DBD156, 500 ms
   "2940RS001N01T01.Unit" : TextRef, internal   // Еденицы измерения При експорте из ECS через скрипт заполняется автоматически, если теги копируются в ручную то требуется задатать свойство Text
   "2940RS001N01T01.Decimals" : TextRef, internal   // Формат отображения При експорте из ECS через скрипт, заполняется автоматически. Если теги копируются в ручную то требуется задатать свойство Text s999999.9
   "2940RS001N01T01.FP_EN.Square" : Bool AT %DB5304.DBX46.0, 500 ms
   "2940RS001N01T01.FP_EN.SquareRoot" : Bool AT %DB5304.DBX46.1, 500 ms
   "2940RS001N01T01.FP_EN.ParentSupress" : Bool AT %DB5304.DBX46.2, 500 ms
   "2940RS001N01T01.FP_EN.ParentSupressUnit" : Bool AT %DB5304.DBX46.3, 500 ms
   "2940RS001N01T01.FP_EN.Force" : Bool AT %DB5304.DBX46.4, 500 ms
   "2940RS001N01T01.FP_EN.Damping" : Bool AT %DB5304.DBX46.5, 500 ms
   "2940RS001N01T01.FP_EN.Gradient_Pos" : Bool AT %DB5304.DBX46.6, 500 ms
   "2940RS001N01T01.FP_EN.Gradient_Neg" : Bool AT %DB5304.DBX46.7, 500 ms
   "2940RS001N01T01.FP_EN.Hysteresis" : Bool AT %DB5304.DBX47.0, 500 ms
   "2940RS001N01T01.FP_EN.Alarm_H3" : Bool AT %DB5304.DBX47.1, 500 ms
   "2940RS001N01T01.FP_EN.Alarm_H2" : Bool AT %DB5304.DBX47.2, 500 ms
   "2940RS001N01T01.FP_EN.Alarm_H1" : Bool AT %DB5304.DBX47.3, 500 ms
   "2940RS001N01T01.FP_EN.Alarm_L1" : Bool AT %DB5304.DBX47.4, 500 ms
   "2940RS001N01T01.FP_EN.Alarm_L2" : Bool AT %DB5304.DBX47.5, 500 ms
   "2940RS001N01T01.FP_EN.Alarm_L3" : Bool AT %DB5304.DBX47.6, 500 ms
   "2940RS001N01T01.FP_EN.AlarmDelay_H3" : Bool AT %DB5304.DBX47.7, 500 ms
   "2940RS001N01T01.FP_EN.AlarmDelay_H2" : Bool AT %DB5304.DBX48.0, 500 ms
   "2940RS001N01T01.FP_EN.AlarmDelay_H1" : Bool AT %DB5304.DBX48.1, 500 ms
   "2940RS001N01T01.FP_EN.AlarmDelay_L1" : Bool AT %DB5304.DBX48.2, 500 ms
   "2940RS001N01T01.FP_EN.AlarmDelay_L2" : Bool AT %DB5304.DBX48.3, 500 ms
   "2940RS001N01T01.FP_EN.AlarmDelay_L3" : Bool AT %DB5304.DBX48.4, 500 ms
   "2940RS001N01T01.FP_EN.ROC_Warn" : Bool AT %DB5304.DBX48.5, 500 ms
   "2940RS001N01T01.FP_EN.U_Range_Warn" : Bool AT %DB5304.DBX48.6, 500 ms
   "2940RS001N01T01.FP_EN.O_Range_Warn" : Bool AT %DB5304.DBX48.7, 500 ms
   "2940RS001N01T01.trend_tag_name" : TextRef, internal   // Еденицы измерения При експорте из ECS через скрипт - заполняется автоматически, если теги копируются в ручную то требуется задатать свойство Text - имя тега для тренда
   "2940RS001N01T01.DQ.AL_H3" : Bool AT %DB5304.DBX16.0, 500 ms
   "2940RS001N01T01.DQ.AL_H2" : Bool AT %DB5304.DBX16.1, 500 ms
   "2940RS001N01T01.DQ.AL_H1" : Bool AT %DB5304.DBX16.2, 500 ms
   "2940RS001N01T01.DQ.AL_L1" : Bool AT %DB5304.DBX16.3, 500 ms
   "2940RS001N01T01.DQ.AL_L2" : Bool AT %DB5304.DBX16.4, 500 ms
   "2940RS001N01T01.DQ.AL_L3" : Bool AT %DB5304.DBX16.5, 500 ms
   "2940RS001N01T01.DQ.SIG_OK" : Bool AT %DB5304.DBX16.6, 500 ms
   "2940RS001N01T01.DQ.LIM_H2" : Bool AT %DB5304.DBX16.7, 500 ms
   "2940RS001N01T01.DQ.LIM_H1" : Bool AT %DB5304.DBX17.0, 500 ms
   "2940RS001N01T01.DQ.LIM_L1" : Bool AT %DB5304.DBX17.1, 500 ms
   "2940RS001N01T01.DQ.LIM_L2" : Bool AT %DB5304.DBX17.2, 500 ms
   "2940RS001N01T01.DQ.GR_P" : Bool AT %DB5304.DBX17.3, 500 ms
   "2940RS001N01T01.DQ.GR_N" : Bool AT %DB5304.DBX17.4, 500 ms
   "2940RS001N01T01.I.IN" : Real AT %DB5304.DBD2, 500 ms
   "2940RS001N01T01.I.SIG_TYPE" : Int AT %DB5304.DBW0, 500 ms
   "2940RS001N01T01.I.FI_BUS" : Byte AT %DB5304.DBB6, 500 ms
   "2940RS001N01T01.DI.U_RANGE" : Bool AT %DB5304.DBX7.0, 500 ms
   "2940RS001N01T01.DI.O_RANGE" : Bool AT %DB5304.DBX7.1, 500 ms
   "2940RS001N01T01.DI.SIG_FAULT" : Bool AT %DB5304.DBX7.2, 500 ms
   "2940RS001N01T01.DI.EnConfig" : Bool AT %DB5304.DBX7.3, 500 ms
   "2940RS001N01T01.DI.AEN" : Bool AT %DB5304.DBX7.4, 500 ms
   "2940RS001N01T01.DI.AL_SUPR" : Bool AT %DB5304.DBX7.5, 500 ms
   "2940RS001N01T01.Q.PV_NORM" : Real AT %DB5304.DBD8, 500 ms
   "2940RS001N01T01.Q.PV_SCAL" : Real AT %DB5304.DBD12, 500 ms
   "2940RS001N01T01.ParentInfo" : TextRef, internal   // Имя родителя для попап окна, вкладка инфо. При експорте из ECS через скрипт заполняется автоматически, если теги копируются в ручную то требуется в ручную задатать свойство Start Value

HMI tags "2080AG500M01"
   "2080AG500M01.AI1" : Real AT %DB4140.DBD6, 500 ms
   "2080AG500M01.AI2" : Real AT %DB4140.DBD10, 500 ms
   "2080AG500M01.AI3" : Real AT %DB4140.DBD14, 500 ms
   "2080AG500M01.AO1a" : Real AT %DB4140.DBD34, 500 ms
   "2080AG500M01.AO1b" : Real AT %DB4140.DBD38, 500 ms
   "2080AG500M01.AO2a" : Real AT %DB4140.DBD42, 500 ms
   "2080AG500M01.AO2b" : Real AT %DB4140.DBD42, 500 ms
   "2080AG500M01.AO3a" : Real AT %DB4140.DBD50, 500 ms
   "2080AG500M01.AO3b" : Real AT %DB4140.DBD46, 500 ms
   "2080AG500M01.BlockInfo" : Array [0..4] of Int AT %DB4140.DBX74.0, 500 ms
   "2080AG500M01.DefaultText" : TextRef, internal   // Заголовок POPUP окна. При експорте из ECS через скрипт заполняется автоматически, если теги копируются в ручную то требуется в ручную задатать свойство Start Value
   "2080AG500M01.DI.ACK" : Bool AT %DB4140.DBX5.3, 500 ms
   "2080AG500M01.DI.ASTR" : Bool AT %DB4140.DBX2.1, 500 ms
   "2080AG500M01.DI.BUSF" : Bool AT %DB4140.DBX4.5, 500 ms
   "2080AG500M01.DI.DIR" : Bool AT %DB4140.DBX2.2, 500 ms
   "2080AG500M01.DI.DOPR" : Bool AT %DB4140.DBX4.6, 500 ms
   "2080AG500M01.DI.DRDY" : Bool AT %DB4140.DBX3.6, 500 ms
   "2080AG500M01.DI.DTEST" : Bool AT %DB4140.DBX4.7, 500 ms
   "2080AG500M01.DI.EARTH" : Bool AT %DB4140.DBX4.1, 500 ms
   "2080AG500M01.DI.ES" : Bool AT %DB4140.DBX5.2, 500 ms
   "2080AG500M01.DI.GFA" : Bool AT %DB4140.DBX4.3, 500 ms
   "2080AG500M01.DI.GWA" : Bool AT %DB4140.DBX4.4, 500 ms
   "2080AG500M01.DI.LSTP" : Bool AT %DB4140.DBX3.2, 500 ms
   "2080AG500M01.DI.LSTR1" : Bool AT %DB4140.DBX3.0, 500 ms
   "2080AG500M01.DI.LSTR2" : Bool AT %DB4140.DBX3.1, 500 ms
   "2080AG500M01.DI.MCC" : Bool AT %DB4140.DBX2.3, 500 ms
   "2080AG500M01.DI.MD" : Bool AT %DB4140.DBX3.7, 500 ms
   "2080AG500M01.DI.OVL" : Bool AT %DB4140.DBX2.5, 500 ms
   "2080AG500M01.DI.RDY" : Bool AT %DB4140.DBX2.4, 500 ms
   "2080AG500M01.DI.REM" : Bool AT %DB4140.DBX3.3, 500 ms
   "2080AG500M01.DI.RET1" : Bool AT %DB4140.DBX2.6, 500 ms
   "2080AG500M01.DI.RET2" : Bool AT %DB4140.DBX2.7, 500 ms
   "2080AG500M01.DI.SEL" : Bool AT %DB4140.DBX2.0, 500 ms
   "2080AG500M01.DI.SFS" : Bool AT %DB4140.DBX5.0, 500 ms
   "2080AG500M01.DI.SLS" : Bool AT %DB4140.DBX5.1, 500 ms
   "2080AG500M01.DI.SSW" : Bool AT %DB4140.DBX3.4, 500 ms
   "2080AG500M01.DI.STALL" : Bool AT %DB4140.DBX4.0, 500 ms
   "2080AG500M01.DI.TFA" : Bool AT %DB4140.DBX3.5, 500 ms
   "2080AG500M01.DI.UBAL" : Bool AT %DB4140.DBX4.2, 500 ms
   "2080AG500M01.DQ.ASTW" : Bool AT %DB4140.DBX32.0, 500 ms
   "2080AG500M01.DQ.AUT" : Bool AT %DB4140.DBX31.4, 500 ms
   "2080AG500M01.DQ.CON1" : Bool AT %DB4140.DBX30.0, 500 ms
   "2080AG500M01.DQ.CON2" : Bool AT %DB4140.DBX30.1, 500 ms
   "2080AG500M01.DQ.LAMP1" : Bool AT %DB4140.DBX30.2, 500 ms
   "2080AG500M01.DQ.LAMP2" : Bool AT %DB4140.DBX30.3, 500 ms
   "2080AG500M01.DQ.LOC" : Bool AT %DB4140.DBX31.2, 500 ms
   "2080AG500M01.DQ.MAN" : Bool AT %DB4140.DBX31.3, 500 ms
   "2080AG500M01.DQ.OK" : Bool AT %DB4140.DBX31.1, 500 ms
   "2080AG500M01.DQ.RD1" : Bool AT %DB4140.DBX30.5, 500 ms
   "2080AG500M01.DQ.RD2" : Bool AT %DB4140.DBX30.6, 500 ms
   "2080AG500M01.DQ.RES" : Bool AT %DB4140.DBX31.6, 500 ms
   "2080AG500M01.DQ.RUN1" : Bool AT %DB4140.DBX30.7, 500 ms
   "2080AG500M01.DQ.RUN2" : Bool AT %DB4140.DBX31.0, 500 ms
   "2080AG500M01.DQ.SACK" : Bool AT %DB4140.DBX30.4, 500 ms
   "2080AG500M01.DQ.SS" : Bool AT %DB4140.DBX31.5, 500 ms
   "2080AG500M01.DQ.TESTP" : Bool AT %DB4140.DBX31.7, 500 ms
   "2080AG500M01.FP_CMD" : Int AT %DB4140.DBW84, 500 ms
   "2080AG500M01.FP_CMD.AckAlarm" : Bool AT %DB4140.DBX84.7, 500 ms
   "2080AG500M01.FP_CMD.Auto" : Bool AT %DB4140.DBX85.0, 500 ms
   "2080AG500M01.FP_CMD.Local" : Bool AT %DB4140.DBX85.2, 500 ms
   "2080AG500M01.FP_CMD.Manual" : Bool AT %DB4140.DBX85.1, 500 ms
   "2080AG500M01.FP_CMD.QuickStop" : Bool AT %DB4140.DBX84.0, 500 ms
   "2080AG500M01.FP_CMD.Reset" : Bool AT %DB4140.DBX85.6, 500 ms
   "2080AG500M01.FP_CMD.Start1" : Bool AT %DB4140.DBX85.3, 500 ms
   "2080AG500M01.FP_CMD.Start2" : Bool AT %DB4140.DBX85.4, 500 ms
   "2080AG500M01.FP_CMD.Stop" : Bool AT %DB4140.DBX85.5, 500 ms
   "2080AG500M01.FP_CMD.Test" : Bool AT %DB4140.DBX85.7, 500 ms
   "2080AG500M01.FP_DIM.Auto" : Bool AT %DB4140.DBX92.0, 500 ms
   "2080AG500M01.FP_DIM.FP_DIM" : Bool AT %DB4140.DBX92.0, 500 ms
   "2080AG500M01.FP_DIM.Local" : Bool AT %DB4140.DBX92.1, 500 ms
   "2080AG500M01.FP_DIM.Manual" : Bool AT %DB4140.DBX92.2, 500 ms
   "2080AG500M01.FP_DIM.QStop" : Bool AT %DB4140.DBX92.7, 500 ms
   "2080AG500M01.FP_DIM.Reset" : Bool AT %DB4140.DBX93.0, 500 ms
   "2080AG500M01.FP_DIM.Start1" : Bool AT %DB4140.DBX92.3, 500 ms
   "2080AG500M01.FP_DIM.Start2" : Bool AT %DB4140.DBX92.4, 500 ms
   "2080AG500M01.FP_DIM.Stop" : Bool AT %DB4140.DBX92.5, 500 ms
   "2080AG500M01.FP_DIM.TEst" : Bool AT %DB4140.DBX92.6, 500 ms
   "2080AG500M01.FP_DIM1" : Array [0..15] of Bool AT %DB4140.DBX92.0, 500 ms
   "2080AG500M01.FP_EN.Mode_Auto" : Bool AT %DB4140.DBX90.0, 500 ms
   "2080AG500M01.FP_EN.Mode_Loc" : Bool AT %DB4140.DBX90.2, 500 ms
   "2080AG500M01.FP_EN.Mode_Loc_1" : Bool AT %DB4140.DBX90.3, 500 ms
   "2080AG500M01.FP_EN.Mode_Man" : Bool AT %DB4140.DBX90.1, 500 ms
   "2080AG500M01.FP_EN.Mode_SS_Field" : Bool AT %DB4140.DBX90.4, 500 ms
   "2080AG500M01.FP_EN.Mode_SS_FP" : Bool AT %DB4140.DBX90.5, 500 ms
   "2080AG500M01.FP_EN.Mode_Test" : Bool AT %DB4140.DBX90.3, 500 ms
   "2080AG500M01.FP_EN.PB_QStop" : Bool AT %DB4140.DBX90.6, 500 ms
   "2080AG500M01.FP_PARM.AI1_Max" : Real AT %DB4140.DBD158, 500 ms
   "2080AG500M01.FP_PARM.AI1_Min" : Real AT %DB4140.DBD162, 500 ms
   "2080AG500M01.FP_PARM.AI2_Max" : Real AT %DB4140.DBD166, 500 ms
   "2080AG500M01.FP_PARM.AI2_Min" : Real AT %DB4140.DBD170, 500 ms
   "2080AG500M01.FP_PARM.AI3_Max" : Real AT %DB4140.DBD174, 500 ms
   "2080AG500M01.FP_PARM.AI3_Min" : Real AT %DB4140.DBD178, 500 ms
   "2080AG500M01.FP_PARM.AO1a_Max" : Real AT %DB4140.DBD182, 500 ms
   "2080AG500M01.FP_PARM.AO1a_Min" : Real AT %DB4140.DBD186, 500 ms
   "2080AG500M01.FP_PARM.AO1b_Max" : Real AT %DB4140.DBD206, 500 ms
   "2080AG500M01.FP_PARM.AO1b_Min" : Real AT %DB4140.DBD210, 500 ms
   "2080AG500M01.FP_PARM.AO2a_Max" : Real AT %DB4140.DBD190, 500 ms
   "2080AG500M01.FP_PARM.AO2a_Min" : Real AT %DB4140.DBD194, 500 ms
   "2080AG500M01.FP_PARM.AO2b_Max" : Real AT %DB4140.DBD214, 500 ms
   "2080AG500M01.FP_PARM.AO2b_Min" : Real AT %DB4140.DBD218, 500 ms
   "2080AG500M01.FP_PARM.AO3a_Max" : Real AT %DB4140.DBD198, 500 ms
   "2080AG500M01.FP_PARM.AO3a_Min" : Real AT %DB4140.DBD202, 500 ms
   "2080AG500M01.FP_PARM.AO3b_Max" : Real AT %DB4140.DBD222, 500 ms
   "2080AG500M01.FP_PARM.AO3b_Min" : Real AT %DB4140.DBD226, 500 ms
   "2080AG500M01.FP_PARM.ChangeDir_Acc" : Int AT %DB4140.DBW138, 500 ms
   "2080AG500M01.FP_PARM.ChangeDir_Pre" : Int AT %DB4140.DBW136, 500 ms
   "2080AG500M01.FP_PARM.DelayStart_Acc" : Int AT %DB4140.DBW114, 500 ms
   "2080AG500M01.FP_PARM.DelayStart_Pre" : Int AT %DB4140.DBW112, 500 ms
   "2080AG500M01.FP_PARM.DelayStop_Acc" : Int AT %DB4140.DBW118, 500 ms
   "2080AG500M01.FP_PARM.DelayStop_Pre" : Int AT %DB4140.DBW116, 500 ms
   "2080AG500M01.FP_PARM.INTL" : Bool AT %DB4140.DBX230.0, 500 ms
   "2080AG500M01.FP_PARM.INTL_SEQ_STP" : Bool AT %DB4140.DBX230.3, 500 ms
   "2080AG500M01.FP_PARM.INTL_SEQ_STR1" : Bool AT %DB4140.DBX230.1, 500 ms
   "2080AG500M01.FP_PARM.INTL_SEQ_STR2" : Bool AT %DB4140.DBX230.2, 500 ms
   "2080AG500M01.FP_PARM.LeaveFS_Acc" : Int AT %DB4140.DBW142, 500 ms
   "2080AG500M01.FP_PARM.LeaveFS_Pre" : Int AT %DB4140.DBW140, 500 ms
   "2080AG500M01.FP_PARM.MD_Freq_PV" : Int AT %DB4140.DBW154, 500 ms
   "2080AG500M01.FP_PARM.MD_Freq_SP" : Int AT %DB4140.DBW152, 500 ms
   "2080AG500M01.FP_PARM.ReachFS_Acc" : Int AT %DB4140.DBW150, 500 ms
   "2080AG500M01.FP_PARM.ReachFS_Pre" : Int AT %DB4140.DBW148, 500 ms
   "2080AG500M01.FP_PARM.ReachLS_Acc" : Int AT %DB4140.DBW146, 500 ms
   "2080AG500M01.FP_PARM.ReachLS_Pre" : Int AT %DB4140.DBW144, 500 ms
   "2080AG500M01.FP_PARM.ReturnMon_Acc" : Int AT %DB4140.DBW122, 500 ms
   "2080AG500M01.FP_PARM.ReturnMon_Pre" : Int AT %DB4140.DBW120, 500 ms
   "2080AG500M01.FP_PARM.RunDelay1_Acc" : Int AT %DB4140.DBW106, 500 ms
   "2080AG500M01.FP_PARM.RunDelay1_Pre" : Int AT %DB4140.DBW104, 500 ms
   "2080AG500M01.FP_PARM.RunDelay2_Acc" : Int AT %DB4140.DBW110, 500 ms
   "2080AG500M01.FP_PARM.RunDelay2_Pre" : Int AT %DB4140.DBW108, 500 ms
   "2080AG500M01.FP_PARM.SpeedMonOffDelay_Acc" : Int AT %DB4140.DBW130, 500 ms
   "2080AG500M01.FP_PARM.SpeedMonOffDelay_Pre" : Int AT %DB4140.DBW128, 500 ms
   "2080AG500M01.FP_PARM.SpeedMonOnDelay_Acc" : Int AT %DB4140.DBW126, 500 ms
   "2080AG500M01.FP_PARM.SpeedMonOnDelay_Pre" : Int AT %DB4140.DBW124, 500 ms
   "2080AG500M01.FP_PARM.SpeedMonTrigDelay_Acc" : Int AT %DB4140.DBW134, 500 ms
   "2080AG500M01.FP_PARM.SpeedMonTrigDelay_Pre" : Int AT %DB4140.DBW132, 500 ms
   "2080AG500M01.FP_PARM.StartWarn_Acc" : Int AT %DB4140.DBW102, 500 ms
   "2080AG500M01.FP_PARM.StartWarn_Pre" : Int AT %DB4140.DBW100, 500 ms
   "2080AG500M01.FP_PARM.StopReason" : Int AT %DB4140.DBW156, 500 ms
   "2080AG500M01.FP_SEL.INCH_Loc" : Bool AT %DB4140.DBX87.7, 500 ms
   "2080AG500M01.FP_SEL.INCH_Man" : Bool AT %DB4140.DBX87.6, 500 ms
   "2080AG500M01.FP_SEL.MD" : Bool AT %DB4140.DBX86.0, 500 ms
   "2080AG500M01.FP_SEL.MD_Maintain" : Bool AT %DB4140.DBX86.3, 500 ms
   "2080AG500M01.FP_SEL.MD_OnOff" : Bool AT %DB4140.DBX86.2, 500 ms
   "2080AG500M01.FP_SEL.MD_Puls" : Bool AT %DB4140.DBX86.1, 500 ms
   "2080AG500M01.FP_SEL.MotorStarter" : Bool AT %DB4140.DBX87.3, 500 ms
   "2080AG500M01.FP_SEL.OutOfSevice" : Bool AT %DB4140.DBX88.0, 500 ms
   "2080AG500M01.FP_SEL.ParentCollection" : Bool AT %DB4140.DBX87.5, 500 ms
   "2080AG500M01.FP_SEL.ParentSupress" : Bool AT %DB4140.DBX87.4, 500 ms
   "2080AG500M01.FP_SEL.STW_AutoStart" : Bool AT %DB4140.DBX86.4, 500 ms
   "2080AG500M01.FP_SEL.STW_Local" : Bool AT %DB4140.DBX86.5, 500 ms
   "2080AG500M01.FP_SEL.STW_Manual" : Bool AT %DB4140.DBX86.6, 500 ms
   "2080AG500M01.FP_SEL.STW_Single" : Bool AT %DB4140.DBX86.7, 500 ms
   "2080AG500M01.FP_SEL.Type_Bimotor" : Bool AT %DB4140.DBX87.1, 500 ms
   "2080AG500M01.FP_SEL.Type_Indication" : Bool AT %DB4140.DBX87.2, 500 ms
   "2080AG500M01.FP_SEL.Type_Unimotor" : Bool AT %DB4140.DBX87.0, 500 ms
   "2080AG500M01.FP_SEL.WarningDrive" : Bool AT %DB4140.DBX88.1, 500 ms
   "2080AG500M01.FP_SHOW.ACK" : Bool AT %DB4140.DBX97.5, 500 ms
   "2080AG500M01.FP_SHOW.AI1" : Bool AT %DB4140.DBX95.0, 500 ms
   "2080AG500M01.FP_SHOW.AI2" : Bool AT %DB4140.DBX95.1, 500 ms
   "2080AG500M01.FP_SHOW.AI3" : Bool AT %DB4140.DBX95.2, 500 ms
   "2080AG500M01.FP_SHOW.ASTR" : Bool AT %DB4140.DBX99.2, 500 ms
   "2080AG500M01.FP_SHOW.B1" : Byte AT %DB4140.DBB95, 500 ms
   "2080AG500M01.FP_SHOW.B2" : Byte AT %DB4140.DBB96, 500 ms
   "2080AG500M01.FP_SHOW.B3" : Byte AT %DB4140.DBB97, 500 ms
   "2080AG500M01.FP_SHOW.B4" : Byte AT %DB4140.DBB98, 500 ms
   "2080AG500M01.FP_SHOW.BUSF" : Bool AT %DB4140.DBX97.2, 500 ms
   "2080AG500M01.FP_SHOW.ChangeDir" : Bool AT %DB4140.DBX99.0, 500 ms
   "2080AG500M01.FP_SHOW.CON2" : Bool AT %DB4140.DBX98.2, 500 ms
   "2080AG500M01.FP_SHOW.DelayRun2" : Bool AT %DB4140.DBX98.7, 500 ms
   "2080AG500M01.FP_SHOW.DOPR" : Bool AT %DB4140.DBX97.3, 500 ms
   "2080AG500M01.FP_SHOW.DRDY" : Bool AT %DB4140.DBX96.4, 500 ms
   "2080AG500M01.FP_SHOW.DTEST" : Bool AT %DB4140.DBX97.4, 500 ms
   "2080AG500M01.FP_SHOW.EARTH" : Bool AT %DB4140.DBX96.6, 500 ms
   "2080AG500M01.FP_SHOW.ES" : Bool AT %DB4140.DBX96.2, 500 ms
   "2080AG500M01.FP_SHOW.GFA" : Bool AT %DB4140.DBX97.0, 500 ms
   "2080AG500M01.FP_SHOW.GWA" : Bool AT %DB4140.DBX97.1, 500 ms
   "2080AG500M01.FP_SHOW.LSTP" : Bool AT %DB4140.DBX95.7, 500 ms
   "2080AG500M01.FP_SHOW.LSTR1" : Bool AT %DB4140.DBX97.6, 500 ms
   "2080AG500M01.FP_SHOW.LSTR2" : Bool AT %DB4140.DBX97.7, 500 ms
   "2080AG500M01.FP_SHOW.MCC" : Bool AT %DB4140.DBX95.4, 500 ms
   "2080AG500M01.FP_SHOW.MD" : Bool AT %DB4140.DBX98.6, 500 ms
   "2080AG500M01.FP_SHOW.OVL" : Bool AT %DB4140.DBX95.6, 500 ms
   "2080AG500M01.FP_SHOW.PB_Auto" : Bool AT %DB4140.DBX94.0, 500 ms
   "2080AG500M01.FP_SHOW.PB_Local" : Bool AT %DB4140.DBX94.1, 500 ms
   "2080AG500M01.FP_SHOW.PB_Manual" : Bool AT %DB4140.DBX94.2, 500 ms
   "2080AG500M01.FP_SHOW.PB_QStop" : Bool AT %DB4140.DBX94.7, 500 ms
   "2080AG500M01.FP_SHOW.PB_Reset" : Bool AT %DB4140.DBX99.1, 500 ms
   "2080AG500M01.FP_SHOW.PB_Start1" : Bool AT %DB4140.DBX94.3, 500 ms
   "2080AG500M01.FP_SHOW.PB_Start2" : Bool AT %DB4140.DBX94.4, 500 ms
   "2080AG500M01.FP_SHOW.PB_Stop" : Bool AT %DB4140.DBX94.5, 500 ms
   "2080AG500M01.FP_SHOW.PB_Test" : Bool AT %DB4140.DBX94.6, 500 ms
   "2080AG500M01.FP_SHOW.RD2" : Bool AT %DB4140.DBX98.3, 500 ms
   "2080AG500M01.FP_SHOW.RDY" : Bool AT %DB4140.DBX95.5, 500 ms
   "2080AG500M01.FP_SHOW.REM" : Bool AT %DB4140.DBX96.0, 500 ms
   "2080AG500M01.FP_SHOW.RET2" : Bool AT %DB4140.DBX98.0, 500 ms
   "2080AG500M01.FP_SHOW.RUN2" : Bool AT %DB4140.DBX98.1, 500 ms
   "2080AG500M01.FP_SHOW.SFS" : Bool AT %DB4140.DBX98.4, 500 ms
   "2080AG500M01.FP_SHOW.SLS" : Bool AT %DB4140.DBX98.5, 500 ms
   "2080AG500M01.FP_SHOW.SP" : Bool AT %DB4140.DBX95.3, 500 ms
   "2080AG500M01.FP_SHOW.SSW" : Bool AT %DB4140.DBX96.1, 500 ms
   "2080AG500M01.FP_SHOW.STALL" : Bool AT %DB4140.DBX96.5, 500 ms
   "2080AG500M01.FP_SHOW.TFA" : Bool AT %DB4140.DBX96.3, 500 ms
   "2080AG500M01.FP_SHOW.UBAL" : Bool AT %DB4140.DBX96.7, 500 ms
   "2080AG500M01.ModePointer" : Int AT %DB4140.DBW496, 500 ms
   "2080AG500M01.MSW" : DWord AT %DB4140.DBD62, 500 ms
   "2080AG500M01.ParentInfo" : TextRef, internal   // Имя родителя для попап окна, вкладка инфо. При експорте из ECS через скрипт заполняется автоматически, если теги копируются в ручную то требуется в ручную задатать свойство Start Value
   "2080AG500M01.SPSET" : Real AT %DB4140.DBD18, 500 ms
   "2080AG500M01.StatusWork" : Int AT %DB4140.DBW494, 500 ms
   "2080AG500M01.STR01" : Byte AT %DB10.DBB64, 500 ms   // Interlock
   "2080AG500M01.STR01.DefaultText" : TextRef, internal
   "2080AG500M01.STR02" : Byte AT %DB10.DBB65, 500 ms   // Interlock
   "2080AG500M01.STR02.DefaultText" : TextRef, internal
   "2080AG500M01.STR03" : Byte AT %DB10.DBB66, 500 ms   // Interlock
   "2080AG500M01.STR03.DefaultText" : TextRef, internal
   "2080AG500M01.STR04" : Byte AT %DB10.DBB67, 500 ms   // Interlock
   "2080AG500M01.STR04.DefaultText" : TextRef, internal
   "2080AG500M01.STR05" : Byte AT %DB10.DBB68, 500 ms   // Interlock
   "2080AG500M01.STR05.DefaultText" : TextRef, internal
   "2080AG500M01.STR06" : Byte AT %DB10.DBB69, 500 ms   // Interlock
   "2080AG500M01.STR06.DefaultText" : TextRef, internal
   "2080AG500M01.STR07" : Byte AT %DB10.DBB70, 500 ms   // Interlock
   "2080AG500M01.STR07.DefaultText" : TextRef, internal
   "2080AG500M01.STR08" : Byte AT %DB10.DBB71, 500 ms   // Interlock
   "2080AG500M01.STR08.DefaultText" : TextRef, internal

HMI tags "2080AG501M01"
   "2080AG501M01.AI1" : Real AT %DB4142.DBD6, 500 ms
   "2080AG501M01.AI2" : Real AT %DB4142.DBD10, 500 ms
   "2080AG501M01.AI3" : Real AT %DB4142.DBD14, 500 ms
   "2080AG501M01.AO1a" : Real AT %DB4142.DBD34, 500 ms
   "2080AG501M01.AO1b" : Real AT %DB4142.DBD38, 500 ms
   "2080AG501M01.AO2a" : Real AT %DB4142.DBD42, 500 ms
   "2080AG501M01.AO2b" : Real AT %DB4142.DBD42, 500 ms
   "2080AG501M01.AO3a" : Real AT %DB4142.DBD50, 500 ms
   "2080AG501M01.AO3b" : Real AT %DB4142.DBD46, 500 ms
   "2080AG501M01.BlockInfo" : Array [0..4] of Int AT %DB4142.DBX74.0, 500 ms
   "2080AG501M01.DefaultText" : TextRef, internal   // Заголовок POPUP окна. При експорте из ECS через скрипт заполняется автоматически, если теги копируются в ручную то требуется в ручную задатать свойство Start Value
   "2080AG501M01.DI.ACK" : Bool AT %DB4142.DBX5.3, 500 ms
   "2080AG501M01.DI.ASTR" : Bool AT %DB4142.DBX2.1, 500 ms
   "2080AG501M01.DI.BUSF" : Bool AT %DB4142.DBX4.5, 500 ms
   "2080AG501M01.DI.DIR" : Bool AT %DB4142.DBX2.2, 500 ms
   "2080AG501M01.DI.DOPR" : Bool AT %DB4142.DBX4.6, 500 ms
   "2080AG501M01.DI.DRDY" : Bool AT %DB4142.DBX3.6, 500 ms
   "2080AG501M01.DI.DTEST" : Bool AT %DB4142.DBX4.7, 500 ms
   "2080AG501M01.DI.EARTH" : Bool AT %DB4142.DBX4.1, 500 ms
   "2080AG501M01.DI.ES" : Bool AT %DB4142.DBX5.2, 500 ms
   "2080AG501M01.DI.GFA" : Bool AT %DB4142.DBX4.3, 500 ms
   "2080AG501M01.DI.GWA" : Bool AT %DB4142.DBX4.4, 500 ms
   "2080AG501M01.DI.LSTP" : Bool AT %DB4142.DBX3.2, 500 ms
   "2080AG501M01.DI.LSTR1" : Bool AT %DB4142.DBX3.0, 500 ms
   "2080AG501M01.DI.LSTR2" : Bool AT %DB4142.DBX3.1, 500 ms
   "2080AG501M01.DI.MCC" : Bool AT %DB4142.DBX2.3, 500 ms
   "2080AG501M01.DI.MD" : Bool AT %DB4142.DBX3.7, 500 ms
   "2080AG501M01.DI.OVL" : Bool AT %DB4142.DBX2.5, 500 ms
   "2080AG501M01.DI.RDY" : Bool AT %DB4142.DBX2.4, 500 ms
   "2080AG501M01.DI.REM" : Bool AT %DB4142.DBX3.3, 500 ms
   "2080AG501M01.DI.RET1" : Bool AT %DB4142.DBX2.6, 500 ms
   "2080AG501M01.DI.RET2" : Bool AT %DB4142.DBX2.7, 500 ms
   "2080AG501M01.DI.SEL" : Bool AT %DB4142.DBX2.0, 500 ms
   "2080AG501M01.DI.SFS" : Bool AT %DB4142.DBX5.0, 500 ms
   "2080AG501M01.DI.SLS" : Bool AT %DB4142.DBX5.1, 500 ms
   "2080AG501M01.DI.SSW" : Bool AT %DB4142.DBX3.4, 500 ms
   "2080AG501M01.DI.STALL" : Bool AT %DB4142.DBX4.0, 500 ms
   "2080AG501M01.DI.TFA" : Bool AT %DB4142.DBX3.5, 500 ms
   "2080AG501M01.DI.UBAL" : Bool AT %DB4142.DBX4.2, 500 ms
   "2080AG501M01.DQ.ASTW" : Bool AT %DB4142.DBX32.0, 500 ms
   "2080AG501M01.DQ.AUT" : Bool AT %DB4142.DBX31.4, 500 ms
   "2080AG501M01.DQ.CON1" : Bool AT %DB4142.DBX30.0, 500 ms
   "2080AG501M01.DQ.CON2" : Bool AT %DB4142.DBX30.1, 500 ms
   "2080AG501M01.DQ.LAMP1" : Bool AT %DB4142.DBX30.2, 500 ms
   "2080AG501M01.DQ.LAMP2" : Bool AT %DB4142.DBX30.3, 500 ms
   "2080AG501M01.DQ.LOC" : Bool AT %DB4142.DBX31.2, 500 ms
   "2080AG501M01.DQ.MAN" : Bool AT %DB4142.DBX31.3, 500 ms
   "2080AG501M01.DQ.OK" : Bool AT %DB4142.DBX31.1, 500 ms
   "2080AG501M01.DQ.RD1" : Bool AT %DB4142.DBX30.5, 500 ms
   "2080AG501M01.DQ.RD2" : Bool AT %DB4142.DBX30.6, 500 ms
   "2080AG501M01.DQ.RES" : Bool AT %DB4142.DBX31.6, 500 ms
   "2080AG501M01.DQ.RUN1" : Bool AT %DB4142.DBX30.7, 500 ms
   "2080AG501M01.DQ.RUN2" : Bool AT %DB4142.DBX31.0, 500 ms
   "2080AG501M01.DQ.SACK" : Bool AT %DB4142.DBX30.4, 500 ms
   "2080AG501M01.DQ.SS" : Bool AT %DB4142.DBX31.5, 500 ms
   "2080AG501M01.DQ.TESTP" : Bool AT %DB4142.DBX31.7, 500 ms
   "2080AG501M01.FP_CMD" : Int AT %DB4142.DBW84, 500 ms
   "2080AG501M01.FP_CMD.AckAlarm" : Bool AT %DB4142.DBX84.7, 500 ms
   "2080AG501M01.FP_CMD.Auto" : Bool AT %DB4142.DBX85.0, 500 ms
   "2080AG501M01.FP_CMD.Local" : Bool AT %DB4142.DBX85.2, 500 ms
   "2080AG501M01.FP_CMD.Manual" : Bool AT %DB4142.DBX85.1, 500 ms
   "2080AG501M01.FP_CMD.QuickStop" : Bool AT %DB4142.DBX84.0, 500 ms
   "2080AG501M01.FP_CMD.Reset" : Bool AT %DB4142.DBX85.6, 500 ms
   "2080AG501M01.FP_CMD.Start1" : Bool AT %DB4142.DBX85.3, 500 ms
   "2080AG501M01.FP_CMD.Start2" : Bool AT %DB4142.DBX85.4, 500 ms
   "2080AG501M01.FP_CMD.Stop" : Bool AT %DB4142.DBX85.5, 500 ms
   "2080AG501M01.FP_CMD.Test" : Bool AT %DB4142.DBX85.7, 500 ms
   "2080AG501M01.FP_DIM.Auto" : Bool AT %DB4142.DBX92.0, 500 ms
   "2080AG501M01.FP_DIM.FP_DIM" : Bool AT %DB4142.DBX92.0, 500 ms
   "2080AG501M01.FP_DIM.Local" : Bool AT %DB4142.DBX92.1, 500 ms
   "2080AG501M01.FP_DIM.Manual" : Bool AT %DB4142.DBX92.2, 500 ms
   "2080AG501M01.FP_DIM.QStop" : Bool AT %DB4142.DBX92.7, 500 ms
   "2080AG501M01.FP_DIM.Reset" : Bool AT %DB4142.DBX93.0, 500 ms
   "2080AG501M01.FP_DIM.Start1" : Bool AT %DB4142.DBX92.3, 500 ms
   "2080AG501M01.FP_DIM.Start2" : Bool AT %DB4142.DBX92.4, 500 ms
   "2080AG501M01.FP_DIM.Stop" : Bool AT %DB4142.DBX92.5, 500 ms
   "2080AG501M01.FP_DIM.TEst" : Bool AT %DB4142.DBX92.6, 500 ms
   "2080AG501M01.FP_DIM1" : Array [0..15] of Bool AT %DB4142.DBX92.0, 500 ms
   "2080AG501M01.FP_EN.Mode_Auto" : Bool AT %DB4142.DBX90.0, 500 ms
   "2080AG501M01.FP_EN.Mode_Loc" : Bool AT %DB4142.DBX90.2, 500 ms
   "2080AG501M01.FP_EN.Mode_Loc_1" : Bool AT %DB4142.DBX90.3, 500 ms
   "2080AG501M01.FP_EN.Mode_Man" : Bool AT %DB4142.DBX90.1, 500 ms
   "2080AG501M01.FP_EN.Mode_SS_Field" : Bool AT %DB4142.DBX90.4, 500 ms
   "2080AG501M01.FP_EN.Mode_SS_FP" : Bool AT %DB4142.DBX90.5, 500 ms
   "2080AG501M01.FP_EN.Mode_Test" : Bool AT %DB4142.DBX90.3, 500 ms
   "2080AG501M01.FP_EN.PB_QStop" : Bool AT %DB4142.DBX90.6, 500 ms
   "2080AG501M01.FP_PARM.AI1_Max" : Real AT %DB4142.DBD158, 500 ms
   "2080AG501M01.FP_PARM.AI1_Min" : Real AT %DB4142.DBD162, 500 ms
   "2080AG501M01.FP_PARM.AI2_Max" : Real AT %DB4142.DBD166, 500 ms
   "2080AG501M01.FP_PARM.AI2_Min" : Real AT %DB4142.DBD170, 500 ms
   "2080AG501M01.FP_PARM.AI3_Max" : Real AT %DB4142.DBD174, 500 ms
   "2080AG501M01.FP_PARM.AI3_Min" : Real AT %DB4142.DBD178, 500 ms
   "2080AG501M01.FP_PARM.AO1a_Max" : Real AT %DB4142.DBD182, 500 ms
   "2080AG501M01.FP_PARM.AO1a_Min" : Real AT %DB4142.DBD186, 500 ms
   "2080AG501M01.FP_PARM.AO1b_Max" : Real AT %DB4142.DBD206, 500 ms
   "2080AG501M01.FP_PARM.AO1b_Min" : Real AT %DB4142.DBD210, 500 ms
   "2080AG501M01.FP_PARM.AO2a_Max" : Real AT %DB4142.DBD190, 500 ms
   "2080AG501M01.FP_PARM.AO2a_Min" : Real AT %DB4142.DBD194, 500 ms
   "2080AG501M01.FP_PARM.AO2b_Max" : Real AT %DB4142.DBD214, 500 ms
   "2080AG501M01.FP_PARM.AO2b_Min" : Real AT %DB4142.DBD218, 500 ms
   "2080AG501M01.FP_PARM.AO3a_Max" : Real AT %DB4142.DBD198, 500 ms
   "2080AG501M01.FP_PARM.AO3a_Min" : Real AT %DB4142.DBD202, 500 ms
   "2080AG501M01.FP_PARM.AO3b_Max" : Real AT %DB4142.DBD222, 500 ms
   "2080AG501M01.FP_PARM.AO3b_Min" : Real AT %DB4142.DBD226, 500 ms
   "2080AG501M01.FP_PARM.ChangeDir_Acc" : Int AT %DB4142.DBW138, 500 ms
   "2080AG501M01.FP_PARM.ChangeDir_Pre" : Int AT %DB4142.DBW136, 500 ms
   "2080AG501M01.FP_PARM.DelayStart_Acc" : Int AT %DB4142.DBW114, 500 ms
   "2080AG501M01.FP_PARM.DelayStart_Pre" : Int AT %DB4142.DBW112, 500 ms
   "2080AG501M01.FP_PARM.DelayStop_Acc" : Int AT %DB4142.DBW118, 500 ms
   "2080AG501M01.FP_PARM.DelayStop_Pre" : Int AT %DB4142.DBW116, 500 ms
   "2080AG501M01.FP_PARM.INTL" : Bool AT %DB4142.DBX230.0, 500 ms
   "2080AG501M01.FP_PARM.INTL_SEQ_STP" : Bool AT %DB4142.DBX230.3, 500 ms
   "2080AG501M01.FP_PARM.INTL_SEQ_STR1" : Bool AT %DB4142.DBX230.1, 500 ms
   "2080AG501M01.FP_PARM.INTL_SEQ_STR2" : Bool AT %DB4142.DBX230.2, 500 ms
   "2080AG501M01.FP_PARM.LeaveFS_Acc" : Int AT %DB4142.DBW142, 500 ms
   "2080AG501M01.FP_PARM.LeaveFS_Pre" : Int AT %DB4142.DBW140, 500 ms
   "2080AG501M01.FP_PARM.MD_Freq_PV" : Int AT %DB4142.DBW154, 500 ms
   "2080AG501M01.FP_PARM.MD_Freq_SP" : Int AT %DB4142.DBW152, 500 ms
   "2080AG501M01.FP_PARM.ReachFS_Acc" : Int AT %DB4142.DBW150, 500 ms
   "2080AG501M01.FP_PARM.ReachFS_Pre" : Int AT %DB4142.DBW148, 500 ms
   "2080AG501M01.FP_PARM.ReachLS_Acc" : Int AT %DB4142.DBW146, 500 ms
   "2080AG501M01.FP_PARM.ReachLS_Pre" : Int AT %DB4142.DBW144, 500 ms
   "2080AG501M01.FP_PARM.ReturnMon_Acc" : Int AT %DB4142.DBW122, 500 ms
   "2080AG501M01.FP_PARM.ReturnMon_Pre" : Int AT %DB4142.DBW120, 500 ms
   "2080AG501M01.FP_PARM.RunDelay1_Acc" : Int AT %DB4142.DBW106, 500 ms
   "2080AG501M01.FP_PARM.RunDelay1_Pre" : Int AT %DB4142.DBW104, 500 ms
   "2080AG501M01.FP_PARM.RunDelay2_Acc" : Int AT %DB4142.DBW110, 500 ms
   "2080AG501M01.FP_PARM.RunDelay2_Pre" : Int AT %DB4142.DBW108, 500 ms
   "2080AG501M01.FP_PARM.SpeedMonOffDelay_Acc" : Int AT %DB4142.DBW130, 500 ms
   "2080AG501M01.FP_PARM.SpeedMonOffDelay_Pre" : Int AT %DB4142.DBW128, 500 ms
   "2080AG501M01.FP_PARM.SpeedMonOnDelay_Acc" : Int AT %DB4142.DBW126, 500 ms
   "2080AG501M01.FP_PARM.SpeedMonOnDelay_Pre" : Int AT %DB4142.DBW124, 500 ms
   "2080AG501M01.FP_PARM.SpeedMonTrigDelay_Acc" : Int AT %DB4142.DBW134, 500 ms
   "2080AG501M01.FP_PARM.SpeedMonTrigDelay_Pre" : Int AT %DB4142.DBW132, 500 ms
   "2080AG501M01.FP_PARM.StartWarn_Acc" : Int AT %DB4142.DBW102, 500 ms
   "2080AG501M01.FP_PARM.StartWarn_Pre" : Int AT %DB4142.DBW100, 500 ms
   "2080AG501M01.FP_PARM.StopReason" : Int AT %DB4142.DBW156, 500 ms
   "2080AG501M01.FP_SEL.INCH_Loc" : Bool AT %DB4142.DBX87.7, 500 ms
   "2080AG501M01.FP_SEL.INCH_Man" : Bool AT %DB4142.DBX87.6, 500 ms
   "2080AG501M01.FP_SEL.MD" : Bool AT %DB4142.DBX86.0, 500 ms
   "2080AG501M01.FP_SEL.MD_Maintain" : Bool AT %DB4142.DBX86.3, 500 ms
   "2080AG501M01.FP_SEL.MD_OnOff" : Bool AT %DB4142.DBX86.2, 500 ms
   "2080AG501M01.FP_SEL.MD_Puls" : Bool AT %DB4142.DBX86.1, 500 ms
   "2080AG501M01.FP_SEL.MotorStarter" : Bool AT %DB4142.DBX87.3, 500 ms
   "2080AG501M01.FP_SEL.OutOfSevice" : Bool AT %DB4142.DBX88.0, 500 ms
   "2080AG501M01.FP_SEL.ParentCollection" : Bool AT %DB4142.DBX87.5, 500 ms
   "2080AG501M01.FP_SEL.ParentSupress" : Bool AT %DB4142.DBX87.4, 500 ms
   "2080AG501M01.FP_SEL.STW_AutoStart" : Bool AT %DB4142.DBX86.4, 500 ms
   "2080AG501M01.FP_SEL.STW_Local" : Bool AT %DB4142.DBX86.5, 500 ms
   "2080AG501M01.FP_SEL.STW_Manual" : Bool AT %DB4142.DBX86.6, 500 ms
   "2080AG501M01.FP_SEL.STW_Single" : Bool AT %DB4142.DBX86.7, 500 ms
   "2080AG501M01.FP_SEL.Type_Bimotor" : Bool AT %DB4142.DBX87.1, 500 ms
   "2080AG501M01.FP_SEL.Type_Indication" : Bool AT %DB4142.DBX87.2, 500 ms
   "2080AG501M01.FP_SEL.Type_Unimotor" : Bool AT %DB4142.DBX87.0, 500 ms
   "2080AG501M01.FP_SEL.WarningDrive" : Bool AT %DB4142.DBX88.1, 500 ms
   "2080AG501M01.FP_SHOW.ACK" : Bool AT %DB4142.DBX97.5, 500 ms
   "2080AG501M01.FP_SHOW.AI1" : Bool AT %DB4142.DBX95.0, 500 ms
   "2080AG501M01.FP_SHOW.AI2" : Bool AT %DB4142.DBX95.1, 500 ms
   "2080AG501M01.FP_SHOW.AI3" : Bool AT %DB4142.DBX95.2, 500 ms
   "2080AG501M01.FP_SHOW.ASTR" : Bool AT %DB4142.DBX99.2, 500 ms
   "2080AG501M01.FP_SHOW.B1" : Byte AT %DB4142.DBB95, 500 ms
   "2080AG501M01.FP_SHOW.B2" : Byte AT %DB4142.DBB96, 500 ms
   "2080AG501M01.FP_SHOW.B3" : Byte AT %DB4142.DBB97, 500 ms
   "2080AG501M01.FP_SHOW.B4" : Byte AT %DB4142.DBB98, 500 ms
   "2080AG501M01.FP_SHOW.BUSF" : Bool AT %DB4142.DBX97.2, 500 ms
   "2080AG501M01.FP_SHOW.ChangeDir" : Bool AT %DB4142.DBX99.0, 500 ms
   "2080AG501M01.FP_SHOW.CON2" : Bool AT %DB4142.DBX98.2, 500 ms
   "2080AG501M01.FP_SHOW.DelayRun2" : Bool AT %DB4142.DBX98.7, 500 ms
   "2080AG501M01.FP_SHOW.DOPR" : Bool AT %DB4142.DBX97.3, 500 ms
   "2080AG501M01.FP_SHOW.DRDY" : Bool AT %DB4142.DBX96.4, 500 ms
   "2080AG501M01.FP_SHOW.DTEST" : Bool AT %DB4142.DBX97.4, 500 ms
   "2080AG501M01.FP_SHOW.EARTH" : Bool AT %DB4142.DBX96.6, 500 ms
   "2080AG501M01.FP_SHOW.ES" : Bool AT %DB4142.DBX96.2, 500 ms
   "2080AG501M01.FP_SHOW.GFA" : Bool AT %DB4142.DBX97.0, 500 ms
   "2080AG501M01.FP_SHOW.GWA" : Bool AT %DB4142.DBX97.1, 500 ms
   "2080AG501M01.FP_SHOW.LSTP" : Bool AT %DB4142.DBX95.7, 500 ms
   "2080AG501M01.FP_SHOW.LSTR1" : Bool AT %DB4142.DBX97.6, 500 ms
   "2080AG501M01.FP_SHOW.LSTR2" : Bool AT %DB4142.DBX97.7, 500 ms
   "2080AG501M01.FP_SHOW.MCC" : Bool AT %DB4142.DBX95.4, 500 ms
   "2080AG501M01.FP_SHOW.MD" : Bool AT %DB4142.DBX98.6, 500 ms
   "2080AG501M01.FP_SHOW.OVL" : Bool AT %DB4142.DBX95.6, 500 ms
   "2080AG501M01.FP_SHOW.PB_Auto" : Bool AT %DB4142.DBX94.0, 500 ms
   "2080AG501M01.FP_SHOW.PB_Local" : Bool AT %DB4142.DBX94.1, 500 ms
   "2080AG501M01.FP_SHOW.PB_Manual" : Bool AT %DB4142.DBX94.2, 500 ms
   "2080AG501M01.FP_SHOW.PB_QStop" : Bool AT %DB4142.DBX94.7, 500 ms
   "2080AG501M01.FP_SHOW.PB_Reset" : Bool AT %DB4142.DBX99.1, 500 ms
   "2080AG501M01.FP_SHOW.PB_Start1" : Bool AT %DB4142.DBX94.3, 500 ms
   "2080AG501M01.FP_SHOW.PB_Start2" : Bool AT %DB4142.DBX94.4, 500 ms
   "2080AG501M01.FP_SHOW.PB_Stop" : Bool AT %DB4142.DBX94.5, 500 ms
   "2080AG501M01.FP_SHOW.PB_Test" : Bool AT %DB4142.DBX94.6, 500 ms
   "2080AG501M01.FP_SHOW.RD2" : Bool AT %DB4142.DBX98.3, 500 ms
   "2080AG501M01.FP_SHOW.RDY" : Bool AT %DB4142.DBX95.5, 500 ms
   "2080AG501M01.FP_SHOW.REM" : Bool AT %DB4142.DBX96.0, 500 ms
   "2080AG501M01.FP_SHOW.RET2" : Bool AT %DB4142.DBX98.0, 500 ms
   "2080AG501M01.FP_SHOW.RUN2" : Bool AT %DB4142.DBX98.1, 500 ms
   "2080AG501M01.FP_SHOW.SFS" : Bool AT %DB4142.DBX98.4, 500 ms
   "2080AG501M01.FP_SHOW.SLS" : Bool AT %DB4142.DBX98.5, 500 ms
   "2080AG501M01.FP_SHOW.SP" : Bool AT %DB4142.DBX95.3, 500 ms
   "2080AG501M01.FP_SHOW.SSW" : Bool AT %DB4142.DBX96.1, 500 ms
   "2080AG501M01.FP_SHOW.STALL" : Bool AT %DB4142.DBX96.5, 500 ms
   "2080AG501M01.FP_SHOW.TFA" : Bool AT %DB4142.DBX96.3, 500 ms
   "2080AG501M01.FP_SHOW.UBAL" : Bool AT %DB4142.DBX96.7, 500 ms
   "2080AG501M01.ModePointer" : Int AT %DB4142.DBW496, 500 ms
   "2080AG501M01.MSW" : DWord AT %DB4142.DBD62, 500 ms
   "2080AG501M01.ParentInfo" : TextRef, internal   // Имя родителя для попап окна, вкладка инфо. При експорте из ECS через скрипт заполняется автоматически, если теги копируются в ручную то требуется в ручную задатать свойство Start Value
   "2080AG501M01.SPSET" : Real AT %DB4142.DBD18, 500 ms
   "2080AG501M01.StatusWork" : Int AT %DB4142.DBW494, 500 ms
   "2080AG501M01.STR01" : Byte AT %DB10.DBB73, 500 ms   // Interlock
   "2080AG501M01.STR01.DefaultText" : TextRef, internal
   "2080AG501M01.STR02" : Byte AT %DB10.DBB74, 500 ms   // Interlock
   "2080AG501M01.STR02.DefaultText" : TextRef, internal
   "2080AG501M01.STR03" : Byte AT %DB10.DBB75, 500 ms   // Interlock
   "2080AG501M01.STR03.DefaultText" : TextRef, internal
   "2080AG501M01.STR04" : Byte AT %DB10.DBB76, 500 ms   // Interlock
   "2080AG501M01.STR04.DefaultText" : TextRef, internal
   "2080AG501M01.STR05" : Byte AT %DB10.DBB77, 500 ms   // Interlock
   "2080AG501M01.STR05.DefaultText" : TextRef, internal
   "2080AG501M01.STR06" : Byte AT %DB10.DBB78, 500 ms   // Interlock
   "2080AG501M01.STR06.DefaultText" : TextRef, internal
   "2080AG501M01.STR07" : Byte AT %DB10.DBB79, 500 ms   // Interlock
   "2080AG501M01.STR07.DefaultText" : TextRef, internal

HMI tags "2080AG502M01"
   "2080AG502M01.AI1" : Real AT %DB4144.DBD6, 500 ms
   "2080AG502M01.AI2" : Real AT %DB4144.DBD10, 500 ms
   "2080AG502M01.AI3" : Real AT %DB4144.DBD14, 500 ms
   "2080AG502M01.AO1a" : Real AT %DB4144.DBD34, 500 ms
   "2080AG502M01.AO1b" : Real AT %DB4144.DBD38, 500 ms
   "2080AG502M01.AO2a" : Real AT %DB4144.DBD42, 500 ms
   "2080AG502M01.AO2b" : Real AT %DB4144.DBD42, 500 ms
   "2080AG502M01.AO3a" : Real AT %DB4144.DBD50, 500 ms
   "2080AG502M01.AO3b" : Real AT %DB4144.DBD46, 500 ms
   "2080AG502M01.BlockInfo" : Array [0..4] of Int AT %DB4144.DBX74.0, 500 ms
   "2080AG502M01.DefaultText" : TextRef, internal   // Заголовок POPUP окна. При експорте из ECS через скрипт заполняется автоматически, если теги копируются в ручную то требуется в ручную задатать свойство Start Value
   "2080AG502M01.DI.ACK" : Bool AT %DB4144.DBX5.3, 500 ms
   "2080AG502M01.DI.ASTR" : Bool AT %DB4144.DBX2.1, 500 ms
   "2080AG502M01.DI.BUSF" : Bool AT %DB4144.DBX4.5, 500 ms
   "2080AG502M01.DI.DIR" : Bool AT %DB4144.DBX2.2, 500 ms
   "2080AG502M01.DI.DOPR" : Bool AT %DB4144.DBX4.6, 500 ms
   "2080AG502M01.DI.DRDY" : Bool AT %DB4144.DBX3.6, 500 ms
   "2080AG502M01.DI.DTEST" : Bool AT %DB4144.DBX4.7, 500 ms
   "2080AG502M01.DI.EARTH" : Bool AT %DB4144.DBX4.1, 500 ms
   "2080AG502M01.DI.ES" : Bool AT %DB4144.DBX5.2, 500 ms
   "2080AG502M01.DI.GFA" : Bool AT %DB4144.DBX4.3, 500 ms
   "2080AG502M01.DI.GWA" : Bool AT %DB4144.DBX4.4, 500 ms
   "2080AG502M01.DI.LSTP" : Bool AT %DB4144.DBX3.2, 500 ms
   "2080AG502M01.DI.LSTR1" : Bool AT %DB4144.DBX3.0, 500 ms
   "2080AG502M01.DI.LSTR2" : Bool AT %DB4144.DBX3.1, 500 ms
   "2080AG502M01.DI.MCC" : Bool AT %DB4144.DBX2.3, 500 ms
   "2080AG502M01.DI.MD" : Bool AT %DB4144.DBX3.7, 500 ms
   "2080AG502M01.DI.OVL" : Bool AT %DB4144.DBX2.5, 500 ms
   "2080AG502M01.DI.RDY" : Bool AT %DB4144.DBX2.4, 500 ms
   "2080AG502M01.DI.REM" : Bool AT %DB4144.DBX3.3, 500 ms
   "2080AG502M01.DI.RET1" : Bool AT %DB4144.DBX2.6, 500 ms
   "2080AG502M01.DI.RET2" : Bool AT %DB4144.DBX2.7, 500 ms
   "2080AG502M01.DI.SEL" : Bool AT %DB4144.DBX2.0, 500 ms
   "2080AG502M01.DI.SFS" : Bool AT %DB4144.DBX5.0, 500 ms
   "2080AG502M01.DI.SLS" : Bool AT %DB4144.DBX5.1, 500 ms
   "2080AG502M01.DI.SSW" : Bool AT %DB4144.DBX3.4, 500 ms
   "2080AG502M01.DI.STALL" : Bool AT %DB4144.DBX4.0, 500 ms
   "2080AG502M01.DI.TFA" : Bool AT %DB4144.DBX3.5, 500 ms
   "2080AG502M01.DI.UBAL" : Bool AT %DB4144.DBX4.2, 500 ms
   "2080AG502M01.DQ.ASTW" : Bool AT %DB4144.DBX32.0, 500 ms
   "2080AG502M01.DQ.AUT" : Bool AT %DB4144.DBX31.4, 500 ms
   "2080AG502M01.DQ.CON1" : Bool AT %DB4144.DBX30.0, 500 ms
   "2080AG502M01.DQ.CON2" : Bool AT %DB4144.DBX30.1, 500 ms
   "2080AG502M01.DQ.LAMP1" : Bool AT %DB4144.DBX30.2, 500 ms
   "2080AG502M01.DQ.LAMP2" : Bool AT %DB4144.DBX30.3, 500 ms
   "2080AG502M01.DQ.LOC" : Bool AT %DB4144.DBX31.2, 500 ms
   "2080AG502M01.DQ.MAN" : Bool AT %DB4144.DBX31.3, 500 ms
   "2080AG502M01.DQ.OK" : Bool AT %DB4144.DBX31.1, 500 ms
   "2080AG502M01.DQ.RD1" : Bool AT %DB4144.DBX30.5, 500 ms
   "2080AG502M01.DQ.RD2" : Bool AT %DB4144.DBX30.6, 500 ms
   "2080AG502M01.DQ.RES" : Bool AT %DB4144.DBX31.6, 500 ms
   "2080AG502M01.DQ.RUN1" : Bool AT %DB4144.DBX30.7, 500 ms
   "2080AG502M01.DQ.RUN2" : Bool AT %DB4144.DBX31.0, 500 ms
   "2080AG502M01.DQ.SACK" : Bool AT %DB4144.DBX30.4, 500 ms
   "2080AG502M01.DQ.SS" : Bool AT %DB4144.DBX31.5, 500 ms
   "2080AG502M01.DQ.TESTP" : Bool AT %DB4144.DBX31.7, 500 ms
   "2080AG502M01.FP_CMD" : Int AT %DB4144.DBW84, 500 ms
   "2080AG502M01.FP_CMD.AckAlarm" : Bool AT %DB4144.DBX84.7, 500 ms
   "2080AG502M01.FP_CMD.Auto" : Bool AT %DB4144.DBX85.0, 500 ms
   "2080AG502M01.FP_CMD.Local" : Bool AT %DB4144.DBX85.2, 500 ms
   "2080AG502M01.FP_CMD.Manual" : Bool AT %DB4144.DBX85.1, 500 ms
   "2080AG502M01.FP_CMD.QuickStop" : Bool AT %DB4144.DBX84.0, 500 ms
   "2080AG502M01.FP_CMD.Reset" : Bool AT %DB4144.DBX85.6, 500 ms
   "2080AG502M01.FP_CMD.Start1" : Bool AT %DB4144.DBX85.3, 500 ms
   "2080AG502M01.FP_CMD.Start2" : Bool AT %DB4144.DBX85.4, 500 ms
   "2080AG502M01.FP_CMD.Stop" : Bool AT %DB4144.DBX85.5, 500 ms
   "2080AG502M01.FP_CMD.Test" : Bool AT %DB4144.DBX85.7, 500 ms
   "2080AG502M01.FP_DIM.Auto" : Bool AT %DB4144.DBX92.0, 500 ms
   "2080AG502M01.FP_DIM.FP_DIM" : Bool AT %DB4144.DBX92.0, 500 ms
   "2080AG502M01.FP_DIM.Local" : Bool AT %DB4144.DBX92.1, 500 ms
   "2080AG502M01.FP_DIM.Manual" : Bool AT %DB4144.DBX92.2, 500 ms
   "2080AG502M01.FP_DIM.QStop" : Bool AT %DB4144.DBX92.7, 500 ms
   "2080AG502M01.FP_DIM.Reset" : Bool AT %DB4144.DBX93.0, 500 ms
   "2080AG502M01.FP_DIM.Start1" : Bool AT %DB4144.DBX92.3, 500 ms
   "2080AG502M01.FP_DIM.Start2" : Bool AT %DB4144.DBX92.4, 500 ms
   "2080AG502M01.FP_DIM.Stop" : Bool AT %DB4144.DBX92.5, 500 ms
   "2080AG502M01.FP_DIM.TEst" : Bool AT %DB4144.DBX92.6, 500 ms
   "2080AG502M01.FP_DIM1" : Array [0..15] of Bool AT %DB4144.DBX92.0, 500 ms
   "2080AG502M01.FP_EN.Mode_Auto" : Bool AT %DB4144.DBX90.0, 500 ms
   "2080AG502M01.FP_EN.Mode_Loc" : Bool AT %DB4144.DBX90.2, 500 ms
   "2080AG502M01.FP_EN.Mode_Loc_1" : Bool AT %DB4144.DBX90.3, 500 ms
   "2080AG502M01.FP_EN.Mode_Man" : Bool AT %DB4144.DBX90.1, 500 ms
   "2080AG502M01.FP_EN.Mode_SS_Field" : Bool AT %DB4144.DBX90.4, 500 ms
   "2080AG502M01.FP_EN.Mode_SS_FP" : Bool AT %DB4144.DBX90.5, 500 ms
   "2080AG502M01.FP_EN.Mode_Test" : Bool AT %DB4144.DBX90.3, 500 ms
   "2080AG502M01.FP_EN.PB_QStop" : Bool AT %DB4144.DBX90.6, 500 ms
   "2080AG502M01.FP_PARM.AI1_Max" : Real AT %DB4144.DBD158, 500 ms
   "2080AG502M01.FP_PARM.AI1_Min" : Real AT %DB4144.DBD162, 500 ms
   "2080AG502M01.FP_PARM.AI2_Max" : Real AT %DB4144.DBD166, 500 ms
   "2080AG502M01.FP_PARM.AI2_Min" : Real AT %DB4144.DBD170, 500 ms
   "2080AG502M01.FP_PARM.AI3_Max" : Real AT %DB4144.DBD174, 500 ms
   "2080AG502M01.FP_PARM.AI3_Min" : Real AT %DB4144.DBD178, 500 ms
   "2080AG502M01.FP_PARM.AO1a_Max" : Real AT %DB4144.DBD182, 500 ms
   "2080AG502M01.FP_PARM.AO1a_Min" : Real AT %DB4144.DBD186, 500 ms
   "2080AG502M01.FP_PARM.AO1b_Max" : Real AT %DB4144.DBD206, 500 ms
   "2080AG502M01.FP_PARM.AO1b_Min" : Real AT %DB4144.DBD210, 500 ms
   "2080AG502M01.FP_PARM.AO2a_Max" : Real AT %DB4144.DBD190, 500 ms
   "2080AG502M01.FP_PARM.AO2a_Min" : Real AT %DB4144.DBD194, 500 ms
   "2080AG502M01.FP_PARM.AO2b_Max" : Real AT %DB4144.DBD214, 500 ms
   "2080AG502M01.FP_PARM.AO2b_Min" : Real AT %DB4144.DBD218, 500 ms
   "2080AG502M01.FP_PARM.AO3a_Max" : Real AT %DB4144.DBD198, 500 ms
   "2080AG502M01.FP_PARM.AO3a_Min" : Real AT %DB4144.DBD202, 500 ms
   "2080AG502M01.FP_PARM.AO3b_Max" : Real AT %DB4144.DBD222, 500 ms
   "2080AG502M01.FP_PARM.AO3b_Min" : Real AT %DB4144.DBD226, 500 ms
   "2080AG502M01.FP_PARM.ChangeDir_Acc" : Int AT %DB4144.DBW138, 500 ms
   "2080AG502M01.FP_PARM.ChangeDir_Pre" : Int AT %DB4144.DBW136, 500 ms
   "2080AG502M01.FP_PARM.DelayStart_Acc" : Int AT %DB4144.DBW114, 500 ms
   "2080AG502M01.FP_PARM.DelayStart_Pre" : Int AT %DB4144.DBW112, 500 ms
   "2080AG502M01.FP_PARM.DelayStop_Acc" : Int AT %DB4144.DBW118, 500 ms
   "2080AG502M01.FP_PARM.DelayStop_Pre" : Int AT %DB4144.DBW116, 500 ms
   "2080AG502M01.FP_PARM.INTL" : Bool AT %DB4144.DBX230.0, 500 ms
   "2080AG502M01.FP_PARM.INTL_SEQ_STP" : Bool AT %DB4144.DBX230.3, 500 ms
   "2080AG502M01.FP_PARM.INTL_SEQ_STR1" : Bool AT %DB4144.DBX230.1, 500 ms
   "2080AG502M01.FP_PARM.INTL_SEQ_STR2" : Bool AT %DB4144.DBX230.2, 500 ms
   "2080AG502M01.FP_PARM.LeaveFS_Acc" : Int AT %DB4144.DBW142, 500 ms
   "2080AG502M01.FP_PARM.LeaveFS_Pre" : Int AT %DB4144.DBW140, 500 ms
   "2080AG502M01.FP_PARM.MD_Freq_PV" : Int AT %DB4144.DBW154, 500 ms
   "2080AG502M01.FP_PARM.MD_Freq_SP" : Int AT %DB4144.DBW152, 500 ms
   "2080AG502M01.FP_PARM.ReachFS_Acc" : Int AT %DB4144.DBW150, 500 ms
   "2080AG502M01.FP_PARM.ReachFS_Pre" : Int AT %DB4144.DBW148, 500 ms
   "2080AG502M01.FP_PARM.ReachLS_Acc" : Int AT %DB4144.DBW146, 500 ms
   "2080AG502M01.FP_PARM.ReachLS_Pre" : Int AT %DB4144.DBW144, 500 ms
   "2080AG502M01.FP_PARM.ReturnMon_Acc" : Int AT %DB4144.DBW122, 500 ms
   "2080AG502M01.FP_PARM.ReturnMon_Pre" : Int AT %DB4144.DBW120, 500 ms
   "2080AG502M01.FP_PARM.RunDelay1_Acc" : Int AT %DB4144.DBW106, 500 ms
   "2080AG502M01.FP_PARM.RunDelay1_Pre" : Int AT %DB4144.DBW104, 500 ms
   "2080AG502M01.FP_PARM.RunDelay2_Acc" : Int AT %DB4144.DBW110, 500 ms
   "2080AG502M01.FP_PARM.RunDelay2_Pre" : Int AT %DB4144.DBW108, 500 ms
   "2080AG502M01.FP_PARM.SpeedMonOffDelay_Acc" : Int AT %DB4144.DBW130, 500 ms
   "2080AG502M01.FP_PARM.SpeedMonOffDelay_Pre" : Int AT %DB4144.DBW128, 500 ms
   "2080AG502M01.FP_PARM.SpeedMonOnDelay_Acc" : Int AT %DB4144.DBW126, 500 ms
   "2080AG502M01.FP_PARM.SpeedMonOnDelay_Pre" : Int AT %DB4144.DBW124, 500 ms
   "2080AG502M01.FP_PARM.SpeedMonTrigDelay_Acc" : Int AT %DB4144.DBW134, 500 ms
   "2080AG502M01.FP_PARM.SpeedMonTrigDelay_Pre" : Int AT %DB4144.DBW132, 500 ms
   "2080AG502M01.FP_PARM.StartWarn_Acc" : Int AT %DB4144.DBW102, 500 ms
   "2080AG502M01.FP_PARM.StartWarn_Pre" : Int AT %DB4144.DBW100, 500 ms
   "2080AG502M01.FP_PARM.StopReason" : Int AT %DB4144.DBW156, 500 ms
   "2080AG502M01.FP_SEL.INCH_Loc" : Bool AT %DB4144.DBX87.7, 500 ms
   "2080AG502M01.FP_SEL.INCH_Man" : Bool AT %DB4144.DBX87.6, 500 ms
   "2080AG502M01.FP_SEL.MD" : Bool AT %DB4144.DBX86.0, 500 ms
   "2080AG502M01.FP_SEL.MD_Maintain" : Bool AT %DB4144.DBX86.3, 500 ms
   "2080AG502M01.FP_SEL.MD_OnOff" : Bool AT %DB4144.DBX86.2, 500 ms
   "2080AG502M01.FP_SEL.MD_Puls" : Bool AT %DB4144.DBX86.1, 500 ms
   "2080AG502M01.FP_SEL.MotorStarter" : Bool AT %DB4144.DBX87.3, 500 ms
   "2080AG502M01.FP_SEL.OutOfSevice" : Bool AT %DB4144.DBX88.0, 500 ms
   "2080AG502M01.FP_SEL.ParentCollection" : Bool AT %DB4144.DBX87.5, 500 ms
   "2080AG502M01.FP_SEL.ParentSupress" : Bool AT %DB4144.DBX87.4, 500 ms
   "2080AG502M01.FP_SEL.STW_AutoStart" : Bool AT %DB4144.DBX86.4, 500 ms
   "2080AG502M01.FP_SEL.STW_Local" : Bool AT %DB4144.DBX86.5, 500 ms
   "2080AG502M01.FP_SEL.STW_Manual" : Bool AT %DB4144.DBX86.6, 500 ms
   "2080AG502M01.FP_SEL.STW_Single" : Bool AT %DB4144.DBX86.7, 500 ms
   "2080AG502M01.FP_SEL.Type_Bimotor" : Bool AT %DB4144.DBX87.1, 500 ms
   "2080AG502M01.FP_SEL.Type_Indication" : Bool AT %DB4144.DBX87.2, 500 ms
   "2080AG502M01.FP_SEL.Type_Unimotor" : Bool AT %DB4144.DBX87.0, 500 ms
   "2080AG502M01.FP_SEL.WarningDrive" : Bool AT %DB4144.DBX88.1, 500 ms
   "2080AG502M01.FP_SHOW.ACK" : Bool AT %DB4144.DBX97.5, 500 ms
   "2080AG502M01.FP_SHOW.AI1" : Bool AT %DB4144.DBX95.0, 500 ms
   "2080AG502M01.FP_SHOW.AI2" : Bool AT %DB4144.DBX95.1, 500 ms
   "2080AG502M01.FP_SHOW.AI3" : Bool AT %DB4144.DBX95.2, 500 ms
   "2080AG502M01.FP_SHOW.ASTR" : Bool AT %DB4144.DBX99.2, 500 ms
   "2080AG502M01.FP_SHOW.B1" : Byte AT %DB4144.DBB95, 500 ms
   "2080AG502M01.FP_SHOW.B2" : Byte AT %DB4144.DBB96, 500 ms
   "2080AG502M01.FP_SHOW.B3" : Byte AT %DB4144.DBB97, 500 ms
   "2080AG502M01.FP_SHOW.B4" : Byte AT %DB4144.DBB98, 500 ms
   "2080AG502M01.FP_SHOW.BUSF" : Bool AT %DB4144.DBX97.2, 500 ms
   "2080AG502M01.FP_SHOW.ChangeDir" : Bool AT %DB4144.DBX99.0, 500 ms
   "2080AG502M01.FP_SHOW.CON2" : Bool AT %DB4144.DBX98.2, 500 ms
   "2080AG502M01.FP_SHOW.DelayRun2" : Bool AT %DB4144.DBX98.7, 500 ms
   "2080AG502M01.FP_SHOW.DOPR" : Bool AT %DB4144.DBX97.3, 500 ms
   "2080AG502M01.FP_SHOW.DRDY" : Bool AT %DB4144.DBX96.4, 500 ms
   "2080AG502M01.FP_SHOW.DTEST" : Bool AT %DB4144.DBX97.4, 500 ms
   "2080AG502M01.FP_SHOW.EARTH" : Bool AT %DB4144.DBX96.6, 500 ms
   "2080AG502M01.FP_SHOW.ES" : Bool AT %DB4144.DBX96.2, 500 ms
   "2080AG502M01.FP_SHOW.GFA" : Bool AT %DB4144.DBX97.0, 500 ms
   "2080AG502M01.FP_SHOW.GWA" : Bool AT %DB4144.DBX97.1, 500 ms
   "2080AG502M01.FP_SHOW.LSTP" : Bool AT %DB4144.DBX95.7, 500 ms
   "2080AG502M01.FP_SHOW.LSTR1" : Bool AT %DB4144.DBX97.6, 500 ms
   "2080AG502M01.FP_SHOW.LSTR2" : Bool AT %DB4144.DBX97.7, 500 ms
   "2080AG502M01.FP_SHOW.MCC" : Bool AT %DB4144.DBX95.4, 500 ms
   "2080AG502M01.FP_SHOW.MD" : Bool AT %DB4144.DBX98.6, 500 ms
   "2080AG502M01.FP_SHOW.OVL" : Bool AT %DB4144.DBX95.6, 500 ms
   "2080AG502M01.FP_SHOW.PB_Auto" : Bool AT %DB4144.DBX94.0, 500 ms
   "2080AG502M01.FP_SHOW.PB_Local" : Bool AT %DB4144.DBX94.1, 500 ms
   "2080AG502M01.FP_SHOW.PB_Manual" : Bool AT %DB4144.DBX94.2, 500 ms
   "2080AG502M01.FP_SHOW.PB_QStop" : Bool AT %DB4144.DBX94.7, 500 ms
   "2080AG502M01.FP_SHOW.PB_Reset" : Bool AT %DB4144.DBX99.1, 500 ms
   "2080AG502M01.FP_SHOW.PB_Start1" : Bool AT %DB4144.DBX94.3, 500 ms
   "2080AG502M01.FP_SHOW.PB_Start2" : Bool AT %DB4144.DBX94.4, 500 ms
   "2080AG502M01.FP_SHOW.PB_Stop" : Bool AT %DB4144.DBX94.5, 500 ms
   "2080AG502M01.FP_SHOW.PB_Test" : Bool AT %DB4144.DBX94.6, 500 ms
   "2080AG502M01.FP_SHOW.RD2" : Bool AT %DB4144.DBX98.3, 500 ms
   "2080AG502M01.FP_SHOW.RDY" : Bool AT %DB4144.DBX95.5, 500 ms
   "2080AG502M01.FP_SHOW.REM" : Bool AT %DB4144.DBX96.0, 500 ms
   "2080AG502M01.FP_SHOW.RET2" : Bool AT %DB4144.DBX98.0, 500 ms
   "2080AG502M01.FP_SHOW.RUN2" : Bool AT %DB4144.DBX98.1, 500 ms
   "2080AG502M01.FP_SHOW.SFS" : Bool AT %DB4144.DBX98.4, 500 ms
   "2080AG502M01.FP_SHOW.SLS" : Bool AT %DB4144.DBX98.5, 500 ms
   "2080AG502M01.FP_SHOW.SP" : Bool AT %DB4144.DBX95.3, 500 ms
   "2080AG502M01.FP_SHOW.SSW" : Bool AT %DB4144.DBX96.1, 500 ms
   "2080AG502M01.FP_SHOW.STALL" : Bool AT %DB4144.DBX96.5, 500 ms
   "2080AG502M01.FP_SHOW.TFA" : Bool AT %DB4144.DBX96.3, 500 ms
   "2080AG502M01.FP_SHOW.UBAL" : Bool AT %DB4144.DBX96.7, 500 ms
   "2080AG502M01.ModePointer" : Int AT %DB4144.DBW496, 500 ms
   "2080AG502M01.MSW" : DWord AT %DB4144.DBD62, 500 ms
   "2080AG502M01.ParentInfo" : TextRef, internal   // Имя родителя для попап окна, вкладка инфо. При експорте из ECS через скрипт заполняется автоматически, если теги копируются в ручную то требуется в ручную задатать свойство Start Value
   "2080AG502M01.SPSET" : Real AT %DB4144.DBD18, 500 ms
   "2080AG502M01.StatusWork" : Int AT %DB4144.DBW494, 500 ms
   "2080AG502M01.STR01" : Byte AT %DB10.DBB81, 500 ms   // Interlock
   "2080AG502M01.STR01.DefaultText" : TextRef, internal
   "2080AG502M01.STR02" : Byte AT %DB10.DBB82, 500 ms   // Interlock
   "2080AG502M01.STR02.DefaultText" : TextRef, internal
   "2080AG502M01.STR03" : Byte AT %DB10.DBB83, 500 ms   // Interlock
   "2080AG502M01.STR03.DefaultText" : TextRef, internal
   "2080AG502M01.STR04" : Byte AT %DB10.DBB84, 500 ms   // Interlock
   "2080AG502M01.STR04.DefaultText" : TextRef, internal
   "2080AG502M01.STR05" : Byte AT %DB10.DBB85, 500 ms   // Interlock
   "2080AG502M01.STR05.DefaultText" : TextRef, internal
   "2080AG502M01.STR06" : Byte AT %DB10.DBB86, 500 ms   // Interlock
   "2080AG502M01.STR06.DefaultText" : TextRef, internal

HMI tags "2080AG503M01"
   "2080AG503M01.AI1" : Real AT %DB4147.DBD6, 500 ms
   "2080AG503M01.AI2" : Real AT %DB4147.DBD10, 500 ms
   "2080AG503M01.AI3" : Real AT %DB4147.DBD14, 500 ms
   "2080AG503M01.AO1a" : Real AT %DB4147.DBD34, 500 ms
   "2080AG503M01.AO1b" : Real AT %DB4147.DBD38, 500 ms
   "2080AG503M01.AO2a" : Real AT %DB4147.DBD42, 500 ms
   "2080AG503M01.AO2b" : Real AT %DB4147.DBD42, 500 ms
   "2080AG503M01.AO3a" : Real AT %DB4147.DBD50, 500 ms
   "2080AG503M01.AO3b" : Real AT %DB4147.DBD46, 500 ms
   "2080AG503M01.BlockInfo" : Array [0..4] of Int AT %DB4147.DBX74.0, 500 ms
   "2080AG503M01.DefaultText" : TextRef, internal   // Заголовок POPUP окна. При експорте из ECS через скрипт заполняется автоматически, если теги копируются в ручную то требуется в ручную задатать свойство Start Value
   "2080AG503M01.DI.ACK" : Bool AT %DB4147.DBX5.3, 500 ms
   "2080AG503M01.DI.ASTR" : Bool AT %DB4147.DBX2.1, 500 ms
   "2080AG503M01.DI.BUSF" : Bool AT %DB4147.DBX4.5, 500 ms
   "2080AG503M01.DI.DIR" : Bool AT %DB4147.DBX2.2, 500 ms
   "2080AG503M01.DI.DOPR" : Bool AT %DB4147.DBX4.6, 500 ms
   "2080AG503M01.DI.DRDY" : Bool AT %DB4147.DBX3.6, 500 ms
   "2080AG503M01.DI.DTEST" : Bool AT %DB4147.DBX4.7, 500 ms
   "2080AG503M01.DI.EARTH" : Bool AT %DB4147.DBX4.1, 500 ms
   "2080AG503M01.DI.ES" : Bool AT %DB4147.DBX5.2, 500 ms
   "2080AG503M01.DI.GFA" : Bool AT %DB4147.DBX4.3, 500 ms
   "2080AG503M01.DI.GWA" : Bool AT %DB4147.DBX4.4, 500 ms
   "2080AG503M01.DI.LSTP" : Bool AT %DB4147.DBX3.2, 500 ms
   "2080AG503M01.DI.LSTR1" : Bool AT %DB4147.DBX3.0, 500 ms
   "2080AG503M01.DI.LSTR2" : Bool AT %DB4147.DBX3.1, 500 ms
   "2080AG503M01.DI.MCC" : Bool AT %DB4147.DBX2.3, 500 ms
   "2080AG503M01.DI.MD" : Bool AT %DB4147.DBX3.7, 500 ms
   "2080AG503M01.DI.OVL" : Bool AT %DB4147.DBX2.5, 500 ms
   "2080AG503M01.DI.RDY" : Bool AT %DB4147.DBX2.4, 500 ms
   "2080AG503M01.DI.REM" : Bool AT %DB4147.DBX3.3, 500 ms
   "2080AG503M01.DI.RET1" : Bool AT %DB4147.DBX2.6, 500 ms
   "2080AG503M01.DI.RET2" : Bool AT %DB4147.DBX2.7, 500 ms
   "2080AG503M01.DI.SEL" : Bool AT %DB4147.DBX2.0, 500 ms
   "2080AG503M01.DI.SFS" : Bool AT %DB4147.DBX5.0, 500 ms
   "2080AG503M01.DI.SLS" : Bool AT %DB4147.DBX5.1, 500 ms
   "2080AG503M01.DI.SSW" : Bool AT %DB4147.DBX3.4, 500 ms
   "2080AG503M01.DI.STALL" : Bool AT %DB4147.DBX4.0, 500 ms
   "2080AG503M01.DI.TFA" : Bool AT %DB4147.DBX3.5, 500 ms
   "2080AG503M01.DI.UBAL" : Bool AT %DB4147.DBX4.2, 500 ms
   "2080AG503M01.DQ.ASTW" : Bool AT %DB4147.DBX32.0, 500 ms
   "2080AG503M01.DQ.AUT" : Bool AT %DB4147.DBX31.4, 500 ms
   "2080AG503M01.DQ.CON1" : Bool AT %DB4147.DBX30.0, 500 ms
   "2080AG503M01.DQ.CON2" : Bool AT %DB4147.DBX30.1, 500 ms
   "2080AG503M01.DQ.LAMP1" : Bool AT %DB4147.DBX30.2, 500 ms
   "2080AG503M01.DQ.LAMP2" : Bool AT %DB4147.DBX30.3, 500 ms
   "2080AG503M01.DQ.LOC" : Bool AT %DB4147.DBX31.2, 500 ms
   "2080AG503M01.DQ.MAN" : Bool AT %DB4147.DBX31.3, 500 ms
   "2080AG503M01.DQ.OK" : Bool AT %DB4147.DBX31.1, 500 ms
   "2080AG503M01.DQ.RD1" : Bool AT %DB4147.DBX30.5, 500 ms
   "2080AG503M01.DQ.RD2" : Bool AT %DB4147.DBX30.6, 500 ms
   "2080AG503M01.DQ.RES" : Bool AT %DB4147.DBX31.6, 500 ms
   "2080AG503M01.DQ.RUN1" : Bool AT %DB4147.DBX30.7, 500 ms
   "2080AG503M01.DQ.RUN2" : Bool AT %DB4147.DBX31.0, 500 ms
   "2080AG503M01.DQ.SACK" : Bool AT %DB4147.DBX30.4, 500 ms
   "2080AG503M01.DQ.SS" : Bool AT %DB4147.DBX31.5, 500 ms
   "2080AG503M01.DQ.TESTP" : Bool AT %DB4147.DBX31.7, 500 ms
   "2080AG503M01.FP_CMD" : Int AT %DB4147.DBW84, 500 ms
   "2080AG503M01.FP_CMD.AckAlarm" : Bool AT %DB4147.DBX84.7, 500 ms
   "2080AG503M01.FP_CMD.Auto" : Bool AT %DB4147.DBX85.0, 500 ms
   "2080AG503M01.FP_CMD.Local" : Bool AT %DB4147.DBX85.2, 500 ms
   "2080AG503M01.FP_CMD.Manual" : Bool AT %DB4147.DBX85.1, 500 ms
   "2080AG503M01.FP_CMD.QuickStop" : Bool AT %DB4147.DBX84.0, 500 ms
   "2080AG503M01.FP_CMD.Reset" : Bool AT %DB4147.DBX85.6, 500 ms
   "2080AG503M01.FP_CMD.Start1" : Bool AT %DB4147.DBX85.3, 500 ms
   "2080AG503M01.FP_CMD.Start2" : Bool AT %DB4147.DBX85.4, 500 ms
   "2080AG503M01.FP_CMD.Stop" : Bool AT %DB4147.DBX85.5, 500 ms
   "2080AG503M01.FP_CMD.Test" : Bool AT %DB4147.DBX85.7, 500 ms
   "2080AG503M01.FP_DIM.Auto" : Bool AT %DB4147.DBX92.0, 500 ms
   "2080AG503M01.FP_DIM.FP_DIM" : Bool AT %DB4147.DBX92.0, 500 ms
   "2080AG503M01.FP_DIM.Local" : Bool AT %DB4147.DBX92.1, 500 ms
   "2080AG503M01.FP_DIM.Manual" : Bool AT %DB4147.DBX92.2, 500 ms
   "2080AG503M01.FP_DIM.QStop" : Bool AT %DB4147.DBX92.7, 500 ms
   "2080AG503M01.FP_DIM.Reset" : Bool AT %DB4147.DBX93.0, 500 ms
   "2080AG503M01.FP_DIM.Start1" : Bool AT %DB4147.DBX92.3, 500 ms
   "2080AG503M01.FP_DIM.Start2" : Bool AT %DB4147.DBX92.4, 500 ms
   "2080AG503M01.FP_DIM.Stop" : Bool AT %DB4147.DBX92.5, 500 ms
   "2080AG503M01.FP_DIM.TEst" : Bool AT %DB4147.DBX92.6, 500 ms
   "2080AG503M01.FP_DIM1" : Array [0..15] of Bool AT %DB4147.DBX92.0, 500 ms
   "2080AG503M01.FP_EN.Mode_Auto" : Bool AT %DB4147.DBX90.0, 500 ms
   "2080AG503M01.FP_EN.Mode_Loc" : Bool AT %DB4147.DBX90.2, 500 ms
   "2080AG503M01.FP_EN.Mode_Loc_1" : Bool AT %DB4147.DBX90.3, 500 ms
   "2080AG503M01.FP_EN.Mode_Man" : Bool AT %DB4147.DBX90.1, 500 ms
   "2080AG503M01.FP_EN.Mode_SS_Field" : Bool AT %DB4147.DBX90.4, 500 ms
   "2080AG503M01.FP_EN.Mode_SS_FP" : Bool AT %DB4147.DBX90.5, 500 ms
   "2080AG503M01.FP_EN.Mode_Test" : Bool AT %DB4147.DBX90.3, 500 ms
   "2080AG503M01.FP_EN.PB_QStop" : Bool AT %DB4147.DBX90.6, 500 ms
   "2080AG503M01.FP_PARM.AI1_Max" : Real AT %DB4147.DBD158, 500 ms
   "2080AG503M01.FP_PARM.AI1_Min" : Real AT %DB4147.DBD162, 500 ms
   "2080AG503M01.FP_PARM.AI2_Max" : Real AT %DB4147.DBD166, 500 ms
   "2080AG503M01.FP_PARM.AI2_Min" : Real AT %DB4147.DBD170, 500 ms
   "2080AG503M01.FP_PARM.AI3_Max" : Real AT %DB4147.DBD174, 500 ms
   "2080AG503M01.FP_PARM.AI3_Min" : Real AT %DB4147.DBD178, 500 ms
   "2080AG503M01.FP_PARM.AO1a_Max" : Real AT %DB4147.DBD182, 500 ms
   "2080AG503M01.FP_PARM.AO1a_Min" : Real AT %DB4147.DBD186, 500 ms
   "2080AG503M01.FP_PARM.AO1b_Max" : Real AT %DB4147.DBD206, 500 ms
   "2080AG503M01.FP_PARM.AO1b_Min" : Real AT %DB4147.DBD210, 500 ms
   "2080AG503M01.FP_PARM.AO2a_Max" : Real AT %DB4147.DBD190, 500 ms
   "2080AG503M01.FP_PARM.AO2a_Min" : Real AT %DB4147.DBD194, 500 ms
   "2080AG503M01.FP_PARM.AO2b_Max" : Real AT %DB4147.DBD214, 500 ms
   "2080AG503M01.FP_PARM.AO2b_Min" : Real AT %DB4147.DBD218, 500 ms
   "2080AG503M01.FP_PARM.AO3a_Max" : Real AT %DB4147.DBD198, 500 ms
   "2080AG503M01.FP_PARM.AO3a_Min" : Real AT %DB4147.DBD202, 500 ms
   "2080AG503M01.FP_PARM.AO3b_Max" : Real AT %DB4147.DBD222, 500 ms
   "2080AG503M01.FP_PARM.AO3b_Min" : Real AT %DB4147.DBD226, 500 ms
   "2080AG503M01.FP_PARM.ChangeDir_Acc" : Int AT %DB4147.DBW138, 500 ms
   "2080AG503M01.FP_PARM.ChangeDir_Pre" : Int AT %DB4147.DBW136, 500 ms
   "2080AG503M01.FP_PARM.DelayStart_Acc" : Int AT %DB4147.DBW114, 500 ms
   "2080AG503M01.FP_PARM.DelayStart_Pre" : Int AT %DB4147.DBW112, 500 ms
   "2080AG503M01.FP_PARM.DelayStop_Acc" : Int AT %DB4147.DBW118, 500 ms
   "2080AG503M01.FP_PARM.DelayStop_Pre" : Int AT %DB4147.DBW116, 500 ms
   "2080AG503M01.FP_PARM.INTL" : Bool AT %DB4147.DBX230.0, 500 ms
   "2080AG503M01.FP_PARM.INTL_SEQ_STP" : Bool AT %DB4147.DBX230.3, 500 ms
   "2080AG503M01.FP_PARM.INTL_SEQ_STR1" : Bool AT %DB4147.DBX230.1, 500 ms
   "2080AG503M01.FP_PARM.INTL_SEQ_STR2" : Bool AT %DB4147.DBX230.2, 500 ms
   "2080AG503M01.FP_PARM.LeaveFS_Acc" : Int AT %DB4147.DBW142, 500 ms
   "2080AG503M01.FP_PARM.LeaveFS_Pre" : Int AT %DB4147.DBW140, 500 ms
   "2080AG503M01.FP_PARM.MD_Freq_PV" : Int AT %DB4147.DBW154, 500 ms
   "2080AG503M01.FP_PARM.MD_Freq_SP" : Int AT %DB4147.DBW152, 500 ms
   "2080AG503M01.FP_PARM.ReachFS_Acc" : Int AT %DB4147.DBW150, 500 ms
   "2080AG503M01.FP_PARM.ReachFS_Pre" : Int AT %DB4147.DBW148, 500 ms
   "2080AG503M01.FP_PARM.ReachLS_Acc" : Int AT %DB4147.DBW146, 500 ms
   "2080AG503M01.FP_PARM.ReachLS_Pre" : Int AT %DB4147.DBW144, 500 ms
   "2080AG503M01.FP_PARM.ReturnMon_Acc" : Int AT %DB4147.DBW122, 500 ms
   "2080AG503M01.FP_PARM.ReturnMon_Pre" : Int AT %DB4147.DBW120, 500 ms
   "2080AG503M01.FP_PARM.RunDelay1_Acc" : Int AT %DB4147.DBW106, 500 ms
   "2080AG503M01.FP_PARM.RunDelay1_Pre" : Int AT %DB4147.DBW104, 500 ms
   "2080AG503M01.FP_PARM.RunDelay2_Acc" : Int AT %DB4147.DBW110, 500 ms
   "2080AG503M01.FP_PARM.RunDelay2_Pre" : Int AT %DB4147.DBW108, 500 ms
   "2080AG503M01.FP_PARM.SpeedMonOffDelay_Acc" : Int AT %DB4147.DBW130, 500 ms
   "2080AG503M01.FP_PARM.SpeedMonOffDelay_Pre" : Int AT %DB4147.DBW128, 500 ms
   "2080AG503M01.FP_PARM.SpeedMonOnDelay_Acc" : Int AT %DB4147.DBW126, 500 ms
   "2080AG503M01.FP_PARM.SpeedMonOnDelay_Pre" : Int AT %DB4147.DBW124, 500 ms
   "2080AG503M01.FP_PARM.SpeedMonTrigDelay_Acc" : Int AT %DB4147.DBW134, 500 ms
   "2080AG503M01.FP_PARM.SpeedMonTrigDelay_Pre" : Int AT %DB4147.DBW132, 500 ms
   "2080AG503M01.FP_PARM.StartWarn_Acc" : Int AT %DB4147.DBW102, 500 ms
   "2080AG503M01.FP_PARM.StartWarn_Pre" : Int AT %DB4147.DBW100, 500 ms
   "2080AG503M01.FP_PARM.StopReason" : Int AT %DB4147.DBW156, 500 ms
   "2080AG503M01.FP_SEL.INCH_Loc" : Bool AT %DB4147.DBX87.7, 500 ms
   "2080AG503M01.FP_SEL.INCH_Man" : Bool AT %DB4147.DBX87.6, 500 ms
   "2080AG503M01.FP_SEL.MD" : Bool AT %DB4147.DBX86.0, 500 ms
   "2080AG503M01.FP_SEL.MD_Maintain" : Bool AT %DB4147.DBX86.3, 500 ms
   "2080AG503M01.FP_SEL.MD_OnOff" : Bool AT %DB4147.DBX86.2, 500 ms
   "2080AG503M01.FP_SEL.MD_Puls" : Bool AT %DB4147.DBX86.1, 500 ms
   "2080AG503M01.FP_SEL.MotorStarter" : Bool AT %DB4147.DBX87.3, 500 ms
   "2080AG503M01.FP_SEL.OutOfSevice" : Bool AT %DB4147.DBX88.0, 500 ms
   "2080AG503M01.FP_SEL.ParentCollection" : Bool AT %DB4147.DBX87.5, 500 ms
   "2080AG503M01.FP_SEL.ParentSupress" : Bool AT %DB4147.DBX87.4, 500 ms
   "2080AG503M01.FP_SEL.STW_AutoStart" : Bool AT %DB4147.DBX86.4, 500 ms
   "2080AG503M01.FP_SEL.STW_Local" : Bool AT %DB4147.DBX86.5, 500 ms
   "2080AG503M01.FP_SEL.STW_Manual" : Bool AT %DB4147.DBX86.6, 500 ms
   "2080AG503M01.FP_SEL.STW_Single" : Bool AT %DB4147.DBX86.7, 500 ms
   "2080AG503M01.FP_SEL.Type_Bimotor" : Bool AT %DB4147.DBX87.1, 500 ms
   "2080AG503M01.FP_SEL.Type_Indication" : Bool AT %DB4147.DBX87.2, 500 ms
   "2080AG503M01.FP_SEL.Type_Unimotor" : Bool AT %DB4147.DBX87.0, 500 ms
   "2080AG503M01.FP_SEL.WarningDrive" : Bool AT %DB4147.DBX88.1, 500 ms
   "2080AG503M01.FP_SHOW.ACK" : Bool AT %DB4147.DBX97.5, 500 ms
   "2080AG503M01.FP_SHOW.AI1" : Bool AT %DB4147.DBX95.0, 500 ms
   "2080AG503M01.FP_SHOW.AI2" : Bool AT %DB4147.DBX95.1, 500 ms
   "2080AG503M01.FP_SHOW.AI3" : Bool AT %DB4147.DBX95.2, 500 ms
   "2080AG503M01.FP_SHOW.ASTR" : Bool AT %DB4147.DBX99.2, 500 ms
   "2080AG503M01.FP_SHOW.B1" : Byte AT %DB4147.DBB95, 500 ms
   "2080AG503M01.FP_SHOW.B2" : Byte AT %DB4147.DBB96, 500 ms
   "2080AG503M01.FP_SHOW.B3" : Byte AT %DB4147.DBB97, 500 ms
   "2080AG503M01.FP_SHOW.B4" : Byte AT %DB4147.DBB98, 500 ms
   "2080AG503M01.FP_SHOW.BUSF" : Bool AT %DB4147.DBX97.2, 500 ms
   "2080AG503M01.FP_SHOW.ChangeDir" : Bool AT %DB4147.DBX99.0, 500 ms
   "2080AG503M01.FP_SHOW.CON2" : Bool AT %DB4147.DBX98.2, 500 ms
   "2080AG503M01.FP_SHOW.DelayRun2" : Bool AT %DB4147.DBX98.7, 500 ms
   "2080AG503M01.FP_SHOW.DOPR" : Bool AT %DB4147.DBX97.3, 500 ms
   "2080AG503M01.FP_SHOW.DRDY" : Bool AT %DB4147.DBX96.4, 500 ms
   "2080AG503M01.FP_SHOW.DTEST" : Bool AT %DB4147.DBX97.4, 500 ms
   "2080AG503M01.FP_SHOW.EARTH" : Bool AT %DB4147.DBX96.6, 500 ms
   "2080AG503M01.FP_SHOW.ES" : Bool AT %DB4147.DBX96.2, 500 ms
   "2080AG503M01.FP_SHOW.GFA" : Bool AT %DB4147.DBX97.0, 500 ms
   "2080AG503M01.FP_SHOW.GWA" : Bool AT %DB4147.DBX97.1, 500 ms
   "2080AG503M01.FP_SHOW.LSTP" : Bool AT %DB4147.DBX95.7, 500 ms
   "2080AG503M01.FP_SHOW.LSTR1" : Bool AT %DB4147.DBX97.6, 500 ms
   "2080AG503M01.FP_SHOW.LSTR2" : Bool AT %DB4147.DBX97.7, 500 ms
   "2080AG503M01.FP_SHOW.MCC" : Bool AT %DB4147.DBX95.4, 500 ms
   "2080AG503M01.FP_SHOW.MD" : Bool AT %DB4147.DBX98.6, 500 ms
   "2080AG503M01.FP_SHOW.OVL" : Bool AT %DB4147.DBX95.6, 500 ms
   "2080AG503M01.FP_SHOW.PB_Auto" : Bool AT %DB4147.DBX94.0, 500 ms
   "2080AG503M01.FP_SHOW.PB_Local" : Bool AT %DB4147.DBX94.1, 500 ms
   "2080AG503M01.FP_SHOW.PB_Manual" : Bool AT %DB4147.DBX94.2, 500 ms
   "2080AG503M01.FP_SHOW.PB_QStop" : Bool AT %DB4147.DBX94.7, 500 ms
   "2080AG503M01.FP_SHOW.PB_Reset" : Bool AT %DB4147.DBX99.1, 500 ms
   "2080AG503M01.FP_SHOW.PB_Start1" : Bool AT %DB4147.DBX94.3, 500 ms
   "2080AG503M01.FP_SHOW.PB_Start2" : Bool AT %DB4147.DBX94.4, 500 ms
   "2080AG503M01.FP_SHOW.PB_Stop" : Bool AT %DB4147.DBX94.5, 500 ms
   "2080AG503M01.FP_SHOW.PB_Test" : Bool AT %DB4147.DBX94.6, 500 ms
   "2080AG503M01.FP_SHOW.RD2" : Bool AT %DB4147.DBX98.3, 500 ms
   "2080AG503M01.FP_SHOW.RDY" : Bool AT %DB4147.DBX95.5, 500 ms
   "2080AG503M01.FP_SHOW.REM" : Bool AT %DB4147.DBX96.0, 500 ms
   "2080AG503M01.FP_SHOW.RET2" : Bool AT %DB4147.DBX98.0, 500 ms
   "2080AG503M01.FP_SHOW.RUN2" : Bool AT %DB4147.DBX98.1, 500 ms
   "2080AG503M01.FP_SHOW.SFS" : Bool AT %DB4147.DBX98.4, 500 ms
   "2080AG503M01.FP_SHOW.SLS" : Bool AT %DB4147.DBX98.5, 500 ms
   "2080AG503M01.FP_SHOW.SP" : Bool AT %DB4147.DBX95.3, 500 ms
   "2080AG503M01.FP_SHOW.SSW" : Bool AT %DB4147.DBX96.1, 500 ms
   "2080AG503M01.FP_SHOW.STALL" : Bool AT %DB4147.DBX96.5, 500 ms
   "2080AG503M01.FP_SHOW.TFA" : Bool AT %DB4147.DBX96.3, 500 ms
   "2080AG503M01.FP_SHOW.UBAL" : Bool AT %DB4147.DBX96.7, 500 ms
   "2080AG503M01.ModePointer" : Int AT %DB4147.DBW496, 500 ms
   "2080AG503M01.MSW" : DWord AT %DB4147.DBD62, 500 ms
   "2080AG503M01.ParentInfo" : TextRef, internal   // Имя родителя для попап окна, вкладка инфо. При експорте из ECS через скрипт заполняется автоматически, если теги копируются в ручную то требуется в ручную задатать свойство Start Value
   "2080AG503M01.SPSET" : Real AT %DB4147.DBD18, 500 ms
   "2080AG503M01.StatusWork" : Int AT %DB4147.DBW494, 500 ms
   "2080AG503M01.STR01" : Byte AT %DB10.DBB97, 500 ms   // Interlock
   "2080AG503M01.STR01.DefaultText" : TextRef, internal
   "2080AG503M01.STR02" : Byte AT %DB10.DBB98, 500 ms   // Interlock
   "2080AG503M01.STR02.DefaultText" : TextRef, internal
   "2080AG503M01.STR03" : Byte AT %DB10.DBB99, 500 ms   // Interlock
   "2080AG503M01.STR03.DefaultText" : TextRef, internal
   "2080AG503M01.STR04" : Byte AT %DB10.DBB100, 500 ms   // Interlock
   "2080AG503M01.STR04.DefaultText" : TextRef, internal
   "2080AG503M01.STR05" : Byte AT %DB10.DBB101, 500 ms   // Interlock
   "2080AG503M01.STR05.DefaultText" : TextRef, internal

